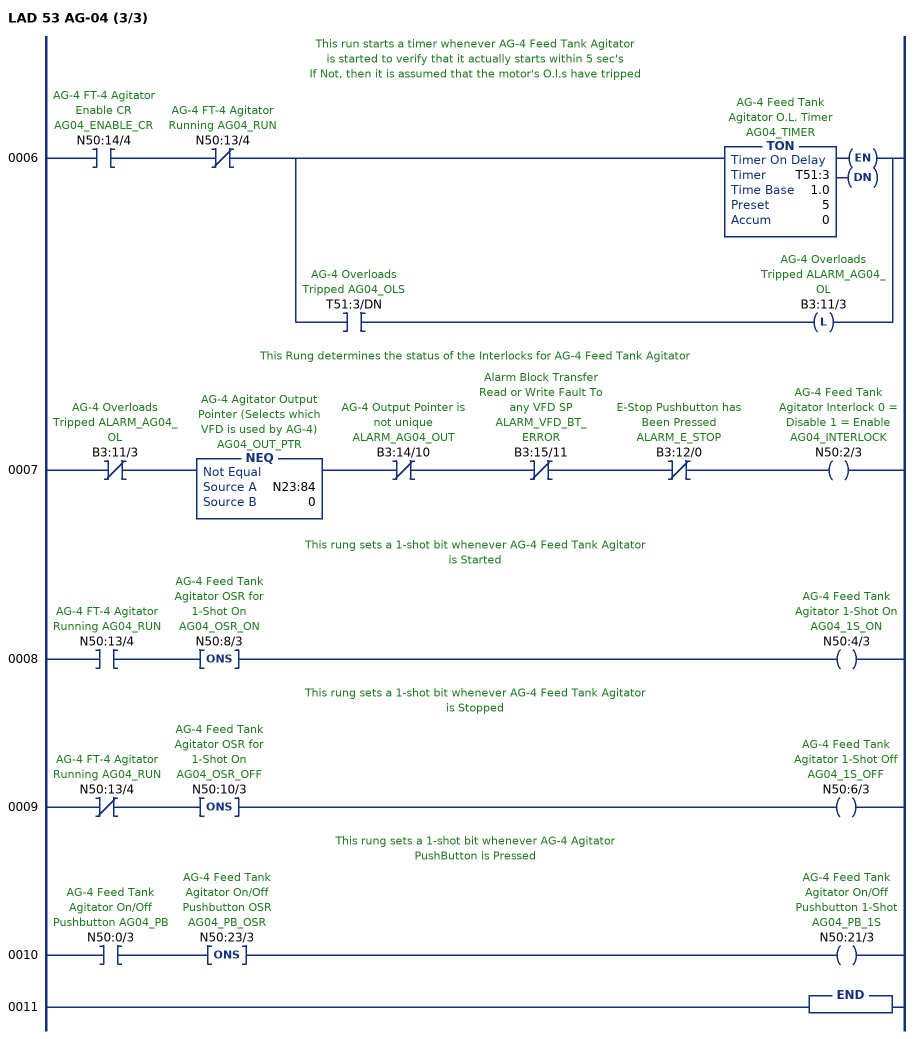
% Rung: 6 %
% This run starts a timer whenever AG-4 Feed Tank Agitator
% is started to verify that it actually starts within 5 sec's
% If Not, then it is assumed that the motor's O.l.s have tripped %
SOR XIC N50:14/4 XIO N50:13/4 BST TON T51:3 1.0 5 0 NXB XIC T51:3/DN OTL B3:11/3 BND EOR
%   N50:14/4  AG04_ENABLE_CR  "AG-4 FT-4 Agitator Enable CR" %
%   N50:13/4  AG04_RUN  "AG-4 FT-4 Agitator Running" %
%   T51:3  AG04_TIMER  "AG-4 Feed Tank Agitator O.L. Timer" %
%   T51:3/DN  AG04_OLS  "AG-4 Overloads Tripped" %
%   B3:11/3  ALARM_AG04_OL  "AG-4 Overloads Tripped" %
% Rung: 7 %
% This Rung determines the status of the Interlocks for AG-4 Feed Tank Agitator %
SOR XIO B3:11/3 NEQ N23:84 0 XIO B3:14/10 XIO B3:15/11 XIO B3:12/0 OTE N50:2/3 EOR
%   B3:11/3  ALARM_AG04_OL  "AG-4 Overloads Tripped" %
%   N23:84  AG04_OUT_PTR  "AG-4 Agitator Output Pointer (Selects which VFD is used by AG-4)" %
%   B3:14/10  ALARM_AG04_OUT  "AG-4 Output Pointer is not unique" %
%   B3:15/11  ALARM_VFD_BT_ERROR  "Alarm Block Transfer Read or Write Fault To any VFD SP" %
%   B3:12/0  ALARM_E_STOP  "E-Stop Pushbutton has Been Pressed" %
%   N50:2/3  AG04_INTERLOCK  "AG-4 Feed Tank Agitator Interlock 0 = Disable 1 = Enable" %
% Rung: 8 %
% This rung sets a 1-shot bit whenever AG-4 Feed Tank Agitator
% is Started %
SOR XIC N50:13/4 OSR N50:8/3 OTE N50:4/3 EOR
%   N50:13/4  AG04_RUN  "AG-4 FT-4 Agitator Running" %
%   N50:8/3  AG04_OSR_ON  "AG-4 Feed Tank Agitator OSR for 1-Shot On" %
%   N50:4/3  AG04_1S_ON  "AG-4 Feed Tank Agitator 1-Shot On" %
% Rung: 9 %
% This rung sets a 1-shot bit whenever AG-4 Feed Tank Agitator
% is Stopped %
SOR XIO N50:13/4 OSR N50:10/3 OTE N50:6/3 EOR
%   N50:13/4  AG04_RUN  "AG-4 FT-4 Agitator Running" %
%   N50:10/3  AG04_OSR_OFF  "AG-4 Feed Tank Agitator OSR for 1-Shot On" %
%   N50:6/3  AG04_1S_OFF  "AG-4 Feed Tank Agitator 1-Shot Off" %
% Rung: 10 %
% This rung sets a 1-shot bit whenever AG-4 Agitator
% PushButton is Pressed %
SOR XIC N50:0/3 OSR N50:23/3 OTE N50:21/3 EOR
%   N50:0/3  AG04_PB  "AG-4 Feed Tank Agitator On/Off Pushbutton" %
%   N50:23/3  AG04_PB_OSR  "AG-4 Feed Tank Agitator On/Off Pushbutton OSR" %
%   N50:21/3  AG04_PB_1S  "AG-4 Feed Tank Agitator On/Off Pushbutton 1-Shot" %
% Rung: 11 %
SOR END EOR

LADDER 56 "VP-09"    % VP-9 Beach-Ross Vacuum Pump Controls %
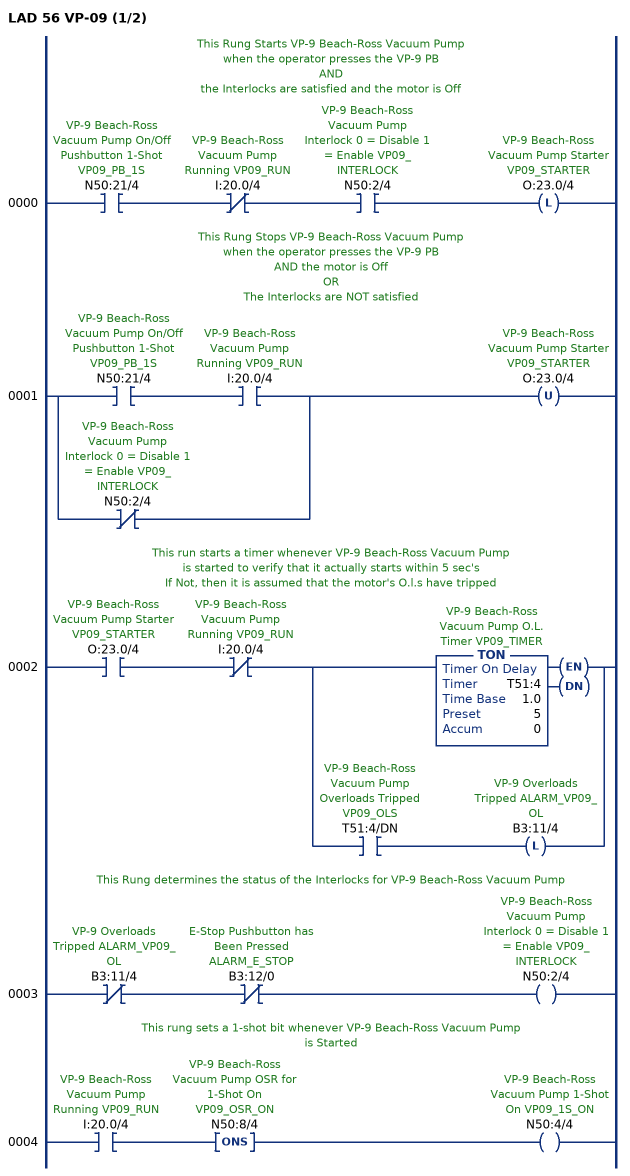
% Rung: 0 %
% This Rung Starts VP-9 Beach-Ross Vacuum Pump
% when the operator presses the VP-9 PB
% AND
% the Interlocks are satisfied and the motor is Off %
SOR XIC N50:21/4 XIO I:20.0/4 XIC N50:2/4 OTL O:23.0/4 EOR
%   N50:21/4  VP09_PB_1S  "VP-9 Beach-Ross Vacuum Pump On/Off Pushbutton 1-Shot" %
%   I:20.0/4  VP09_RUN  "VP-9 Beach-Ross Vacuum Pump Running" %
%   N50:2/4  VP09_INTERLOCK  "VP-9 Beach-Ross Vacuum Pump Interlock 0 = Disable 1 = Enable" %
%   O:23.0/4  VP09_STARTER  "VP-9 Beach-Ross Vacuum Pump Starter" %
% Rung: 1 %
% This Rung Stops VP-9 Beach-Ross Vacuum Pump
% when the operator presses the VP-9 PB
% AND the motor is Off
% OR
% The Interlocks are NOT satisfied %
SOR BST XIC N50:21/4 XIC I:20.0/4 NXB XIO N50:2/4 BND OTU O:23.0/4 EOR
%   N50:21/4  VP09_PB_1S  "VP-9 Beach-Ross Vacuum Pump On/Off Pushbutton 1-Shot" %
%   I:20.0/4  VP09_RUN  "VP-9 Beach-Ross Vacuum Pump Running" %
%   N50:2/4  VP09_INTERLOCK  "VP-9 Beach-Ross Vacuum Pump Interlock 0 = Disable 1 = Enable" %
%   O:23.0/4  VP09_STARTER  "VP-9 Beach-Ross Vacuum Pump Starter" %
% Rung: 2 %
% This run starts a timer whenever VP-9 Beach-Ross Vacuum Pump
% is started to verify that it actually starts within 5 sec's
% If Not, then it is assumed that the motor's O.l.s have tripped %
SOR XIC O:23.0/4 XIO I:20.0/4 BST TON T51:4 1.0 5 0 NXB XIC T51:4/DN OTL B3:11/4 BND EOR
%   O:23.0/4  VP09_STARTER  "VP-9 Beach-Ross Vacuum Pump Starter" %
%   I:20.0/4  VP09_RUN  "VP-9 Beach-Ross Vacuum Pump Running" %
%   T51:4  VP09_TIMER  "VP-9 Beach-Ross Vacuum Pump O.L. Timer" %
%   T51:4/DN  VP09_OLS  "VP-9 Beach-Ross Vacuum Pump Overloads Tripped" %
%   B3:11/4  ALARM_VP09_OL  "VP-9 Overloads Tripped" %
% Rung: 3 %
% This Rung determines the status of the Interlocks for VP-9 Beach-Ross Vacuum Pump %
SOR XIO B3:11/4 XIO B3:12/0 OTE N50:2/4 EOR
%   B3:11/4  ALARM_VP09_OL  "VP-9 Overloads Tripped" %
%   B3:12/0  ALARM_E_STOP  "E-Stop Pushbutton has Been Pressed" %
%   N50:2/4  VP09_INTERLOCK  "VP-9 Beach-Ross Vacuum Pump Interlock 0 = Disable 1 = Enable" %
% Rung: 4 %
% This rung sets a 1-shot bit whenever VP-9 Beach-Ross Vacuum Pump
% is Started %
SOR XIC I:20.0/4 OSR N50:8/4 OTE N50:4/4 EOR
%   I:20.0/4  VP09_RUN  "VP-9 Beach-Ross Vacuum Pump Running" %
%   N50:8/4  VP09_OSR_ON  "VP-9 Beach-Ross Vacuum Pump OSR for 1-Shot On" %
%   N50:4/4  VP09_1S_ON  "VP-9 Beach-Ross Vacuum Pump 1-Shot On" %

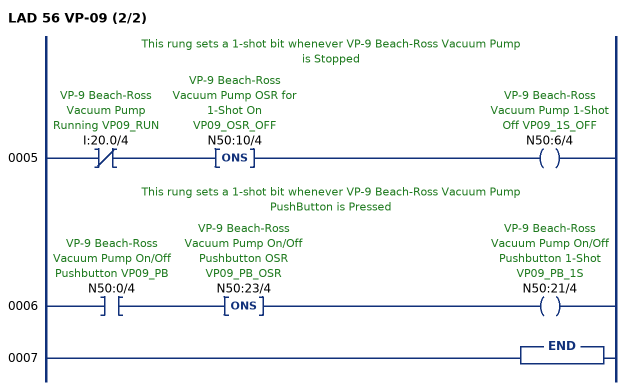
% Rung: 5 %
% This rung sets a 1-shot bit whenever VP-9 Beach-Ross Vacuum Pump
% is Stopped %
SOR XIO I:20.0/4 OSR N50:10/4 OTE N50:6/4 EOR
%   I:20.0/4  VP09_RUN  "VP-9 Beach-Ross Vacuum Pump Running" %
%   N50:10/4  VP09_OSR_OFF  "VP-9 Beach-Ross Vacuum Pump OSR for 1-Shot On" %
%   N50:6/4  VP09_1S_OFF  "VP-9 Beach-Ross Vacuum Pump 1-Shot Off" %
% Rung: 6 %
% This rung sets a 1-shot bit whenever VP-9 Beach-Ross Vacuum Pump
% PushButton is Pressed %
SOR XIC N50:0/4 OSR N50:23/4 OTE N50:21/4 EOR
%   N50:0/4  VP09_PB  "VP-9 Beach-Ross Vacuum Pump On/Off Pushbutton" %
%   N50:23/4  VP09_PB_OSR  "VP-9 Beach-Ross Vacuum Pump On/Off Pushbutton OSR" %
%   N50:21/4  VP09_PB_1S  "VP-9 Beach-Ross Vacuum Pump On/Off Pushbutton 1-Shot" %
% Rung: 7 %
SOR END EOR

LADDER 57 "VP-10"    % VP-10 Kinney Vacuum Pump Controls %
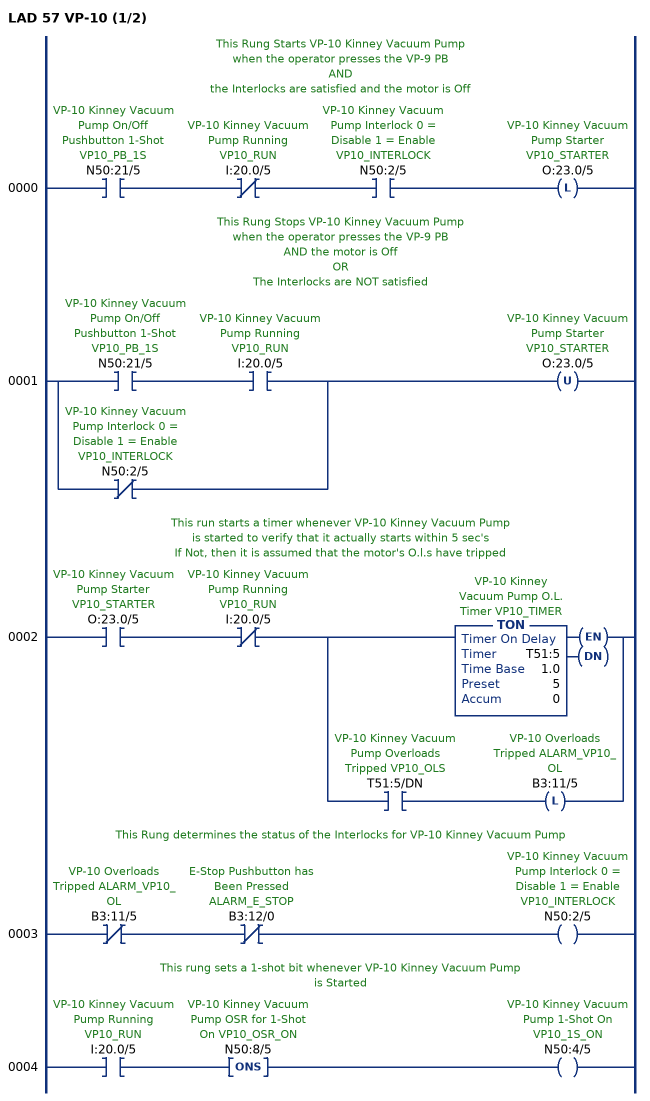
% Rung: 0 %
% This Rung Starts VP-10 Kinney Vacuum Pump
% when the operator presses the VP-9 PB
% AND
% the Interlocks are satisfied and the motor is Off %
SOR XIC N50:21/5 XIO I:20.0/5 XIC N50:2/5 OTL O:23.0/5 EOR
%   N50:21/5  VP10_PB_1S  "VP-10 Kinney Vacuum Pump On/Off Pushbutton 1-Shot" %
%   I:20.0/5  VP10_RUN  "VP-10 Kinney Vacuum Pump Running" %
%   N50:2/5  VP10_INTERLOCK  "VP-10 Kinney Vacuum Pump Interlock 0 = Disable 1 = Enable" %
%   O:23.0/5  VP10_STARTER  "VP-10 Kinney Vacuum Pump Starter" %
% Rung: 1 %
% This Rung Stops VP-10 Kinney Vacuum Pump
% when the operator presses the VP-9 PB
% AND the motor is Off
% OR
% The Interlocks are NOT satisfied %
SOR BST XIC N50:21/5 XIC I:20.0/5 NXB XIO N50:2/5 BND OTU O:23.0/5 EOR
%   N50:21/5  VP10_PB_1S  "VP-10 Kinney Vacuum Pump On/Off Pushbutton 1-Shot" %
%   I:20.0/5  VP10_RUN  "VP-10 Kinney Vacuum Pump Running" %
%   N50:2/5  VP10_INTERLOCK  "VP-10 Kinney Vacuum Pump Interlock 0 = Disable 1 = Enable" %
%   O:23.0/5  VP10_STARTER  "VP-10 Kinney Vacuum Pump Starter" %
% Rung: 2 %
% This run starts a timer whenever VP-10 Kinney Vacuum Pump
% is started to verify that it actually starts within 5 sec's
% If Not, then it is assumed that the motor's O.l.s have tripped %
SOR XIC O:23.0/5 XIO I:20.0/5 BST TON T51:5 1.0 5 0 NXB XIC T51:5/DN OTL B3:11/5 BND EOR
%   O:23.0/5  VP10_STARTER  "VP-10 Kinney Vacuum Pump Starter" %
%   I:20.0/5  VP10_RUN  "VP-10 Kinney Vacuum Pump Running" %
%   T51:5  VP10_TIMER  "VP-10 Kinney Vacuum Pump O.L. Timer" %
%   T51:5/DN  VP10_OLS  "VP-10 Kinney Vacuum Pump Overloads Tripped" %
%   B3:11/5  ALARM_VP10_OL  "VP-10 Overloads Tripped" %
% Rung: 3 %
% This Rung determines the status of the Interlocks for VP-10 Kinney Vacuum Pump %
SOR XIO B3:11/5 XIO B3:12/0 OTE N50:2/5 EOR
%   B3:11/5  ALARM_VP10_OL  "VP-10 Overloads Tripped" %
%   B3:12/0  ALARM_E_STOP  "E-Stop Pushbutton has Been Pressed" %
%   N50:2/5  VP10_INTERLOCK  "VP-10 Kinney Vacuum Pump Interlock 0 = Disable 1 = Enable" %
% Rung: 4 %
% This rung sets a 1-shot bit whenever VP-10 Kinney Vacuum Pump
% is Started %
SOR XIC I:20.0/5 OSR N50:8/5 OTE N50:4/5 EOR
%   I:20.0/5  VP10_RUN  "VP-10 Kinney Vacuum Pump Running" %
%   N50:8/5  VP10_OSR_ON  "VP-10 Kinney Vacuum Pump OSR for 1-Shot On" %
%   N50:4/5  VP10_1S_ON  "VP-10 Kinney Vacuum Pump 1-Shot On" %

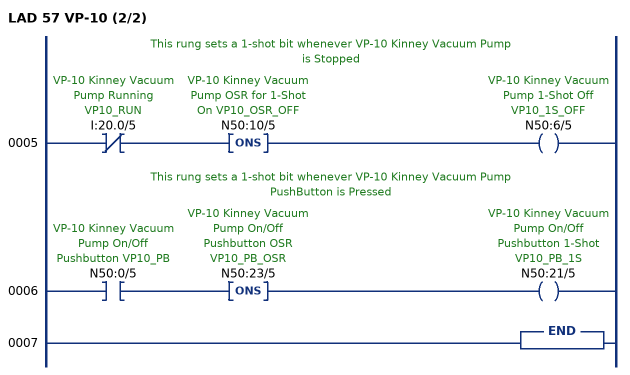
% Rung: 5 %
% This rung sets a 1-shot bit whenever VP-10 Kinney Vacuum Pump
% is Stopped %
SOR XIO I:20.0/5 OSR N50:10/5 OTE N50:6/5 EOR
%   I:20.0/5  VP10_RUN  "VP-10 Kinney Vacuum Pump Running" %
%   N50:10/5  VP10_OSR_OFF  "VP-10 Kinney Vacuum Pump OSR for 1-Shot On" %
%   N50:6/5  VP10_1S_OFF  "VP-10 Kinney Vacuum Pump 1-Shot Off" %
% Rung: 6 %
% This rung sets a 1-shot bit whenever VP-10 Kinney Vacuum Pump
% PushButton is Pressed %
SOR XIC N50:0/5 OSR N50:23/5 OTE N50:21/5 EOR
%   N50:0/5  VP10_PB  "VP-10 Kinney Vacuum Pump On/Off Pushbutton" %
%   N50:23/5  VP10_PB_OSR  "VP-10 Kinney Vacuum Pump On/Off Pushbutton OSR" %
%   N50:21/5  VP10_PB_1S  "VP-10 Kinney Vacuum Pump On/Off Pushbutton 1-Shot" %
% Rung: 7 %
SOR END EOR

LADDER 60 "PU-11"    % PU-11 Tempered Water Loop No-1 Circ Pump Controls %
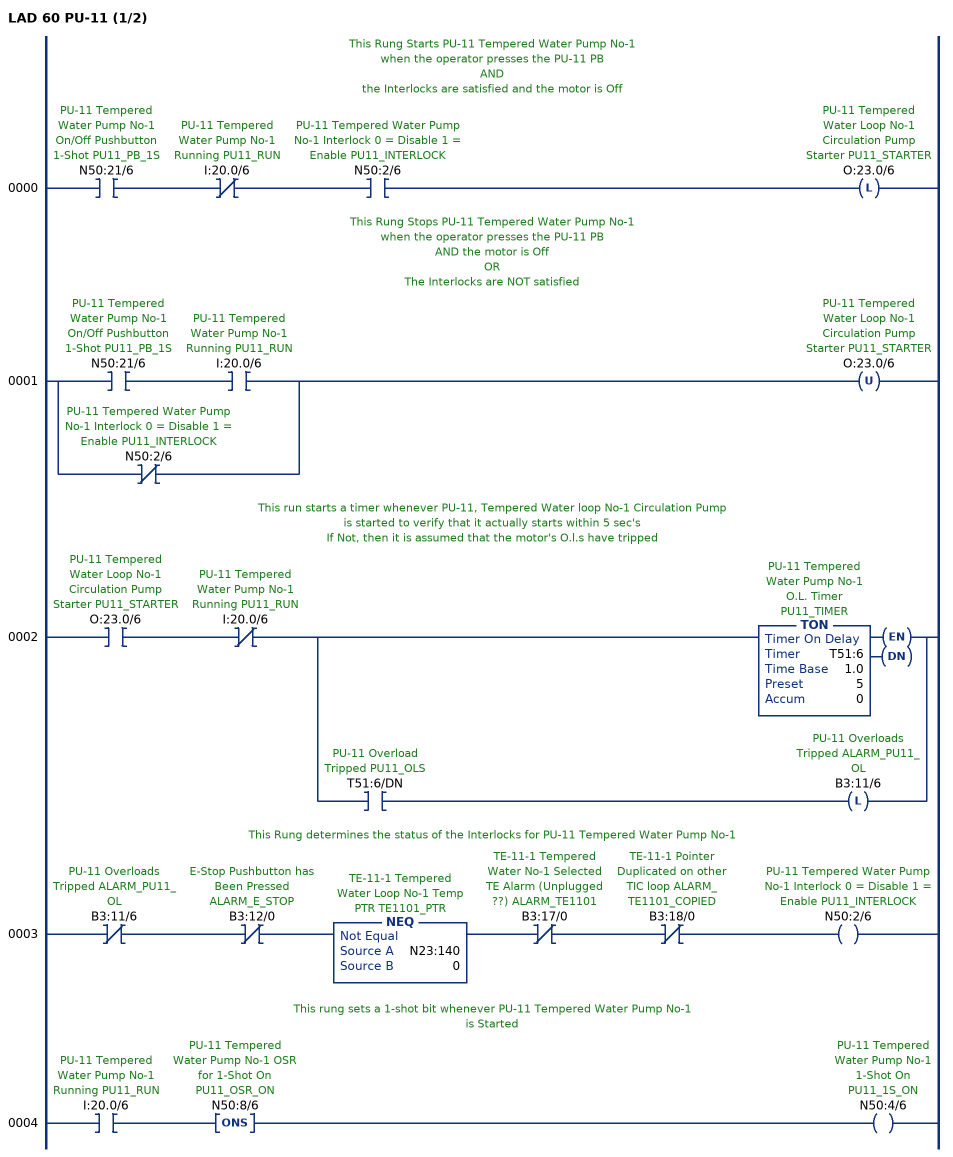
% Rung: 0 %
% This Rung Starts PU-11 Tempered Water Pump No-1
% when the operator presses the PU-11 PB
% AND
% the Interlocks are satisfied and the motor is Off %
SOR XIC N50:21/6 XIO I:20.0/6 XIC N50:2/6 OTL O:23.0/6 EOR
%   N50:21/6  PU11_PB_1S  "PU-11 Tempered Water Pump No-1 On/Off Pushbutton 1-Shot" %
%   I:20.0/6  PU11_RUN  "PU-11 Tempered Water Pump No-1 Running" %
%   N50:2/6  PU11_INTERLOCK  "PU-11 Tempered Water Pump No-1 Interlock 0 = Disable 1 = Enable" %
%   O:23.0/6  PU11_STARTER  "PU-11 Tempered Water Loop No-1 Circulation Pump Starter" %
% Rung: 1 %
% This Rung Stops PU-11 Tempered Water Pump No-1
% when the operator presses the PU-11 PB
% AND the motor is Off
% OR
% The Interlocks are NOT satisfied %
SOR BST XIC N50:21/6 XIC I:20.0/6 NXB XIO N50:2/6 BND OTU O:23.0/6 EOR
%   N50:21/6  PU11_PB_1S  "PU-11 Tempered Water Pump No-1 On/Off Pushbutton 1-Shot" %
%   I:20.0/6  PU11_RUN  "PU-11 Tempered Water Pump No-1 Running" %
%   N50:2/6  PU11_INTERLOCK  "PU-11 Tempered Water Pump No-1 Interlock 0 = Disable 1 = Enable" %
%   O:23.0/6  PU11_STARTER  "PU-11 Tempered Water Loop No-1 Circulation Pump Starter" %
% Rung: 2 %
% This run starts a timer whenever PU-11, Tempered Water loop No-1 Circulation Pump
% is started to verify that it actually starts within 5 sec's
% If Not, then it is assumed that the motor's O.l.s have tripped %
SOR XIC O:23.0/6 XIO I:20.0/6 BST TON T51:6 1.0 5 0 NXB XIC T51:6/DN OTL B3:11/6 BND EOR
%   O:23.0/6  PU11_STARTER  "PU-11 Tempered Water Loop No-1 Circulation Pump Starter" %
%   I:20.0/6  PU11_RUN  "PU-11 Tempered Water Pump No-1 Running" %
%   T51:6  PU11_TIMER  "PU-11 Tempered Water Pump No-1 O.L. Timer" %
%   T51:6/DN  PU11_OLS  "PU-11 Overload Tripped" %
%   B3:11/6  ALARM_PU11_OL  "PU-11 Overloads Tripped" %
% Rung: 3 %
% This Rung determines the status of the Interlocks for PU-11 Tempered Water Pump No-1 %
SOR XIO B3:11/6 XIO B3:12/0 NEQ N23:140 0 XIO B3:17/0 XIO B3:18/0 OTE N50:2/6 EOR
%   B3:11/6  ALARM_PU11_OL  "PU-11 Overloads Tripped" %
%   B3:12/0  ALARM_E_STOP  "E-Stop Pushbutton has Been Pressed" %
%   N23:140  TE1101_PTR  "TE-11-1 Tempered Water Loop No-1 Temp PTR" %
%   B3:17/0  ALARM_TE1101  "TE-11-1 Tempered Water No-1 Selected TE Alarm (Unplugged ??)" %
%   B3:18/0  ALARM_TE1101_COPIED  "TE-11-1 Pointer Duplicated on other TIC loop" %
%   N50:2/6  PU11_INTERLOCK  "PU-11 Tempered Water Pump No-1 Interlock 0 = Disable 1 = Enable" %
% Rung: 4 %
% This rung sets a 1-shot bit whenever PU-11 Tempered Water Pump No-1
% is Started %
SOR XIC I:20.0/6 OSR N50:8/6 OTE N50:4/6 EOR
%   I:20.0/6  PU11_RUN  "PU-11 Tempered Water Pump No-1 Running" %
%   N50:8/6  PU11_OSR_ON  "PU-11 Tempered Water Pump No-1 OSR for 1-Shot On" %
%   N50:4/6  PU11_1S_ON  "PU-11 Tempered Water Pump No-1 1-Shot On" %

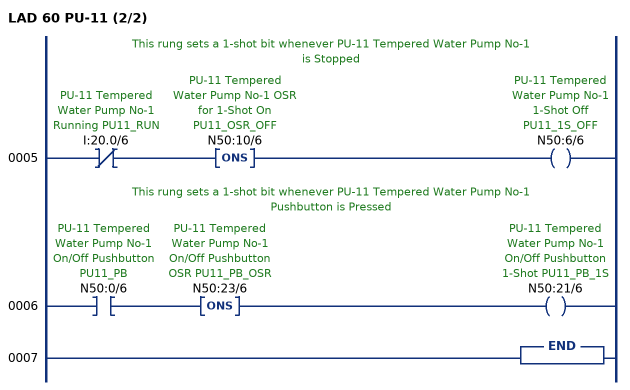
% Rung: 5 %
% This rung sets a 1-shot bit whenever PU-11 Tempered Water Pump No-1
% is Stopped %
SOR XIO I:20.0/6 OSR N50:10/6 OTE N50:6/6 EOR
%   I:20.0/6  PU11_RUN  "PU-11 Tempered Water Pump No-1 Running" %
%   N50:10/6  PU11_OSR_OFF  "PU-11 Tempered Water Pump No-1 OSR for 1-Shot On" %
%   N50:6/6  PU11_1S_OFF  "PU-11 Tempered Water Pump No-1 1-Shot Off" %
% Rung: 6 %
% This rung sets a 1-shot bit whenever PU-11 Tempered Water Pump No-1
% Pushbutton is Pressed %
SOR XIC N50:0/6 OSR N50:23/6 OTE N50:21/6 EOR
%   N50:0/6  PU11_PB  "PU-11 Tempered Water Pump No-1 On/Off Pushbutton" %
%   N50:23/6  PU11_PB_OSR  "PU-11 Tempered Water Pump No-1 On/Off Pushbutton OSR" %
%   N50:21/6  PU11_PB_1S  "PU-11 Tempered Water Pump No-1 On/Off Pushbutton 1-Shot" %
% Rung: 7 %
SOR END EOR

LADDER 61 "PU-12"    % PU-12 Tempered Water Loop No-2 Circ Pump Controls %
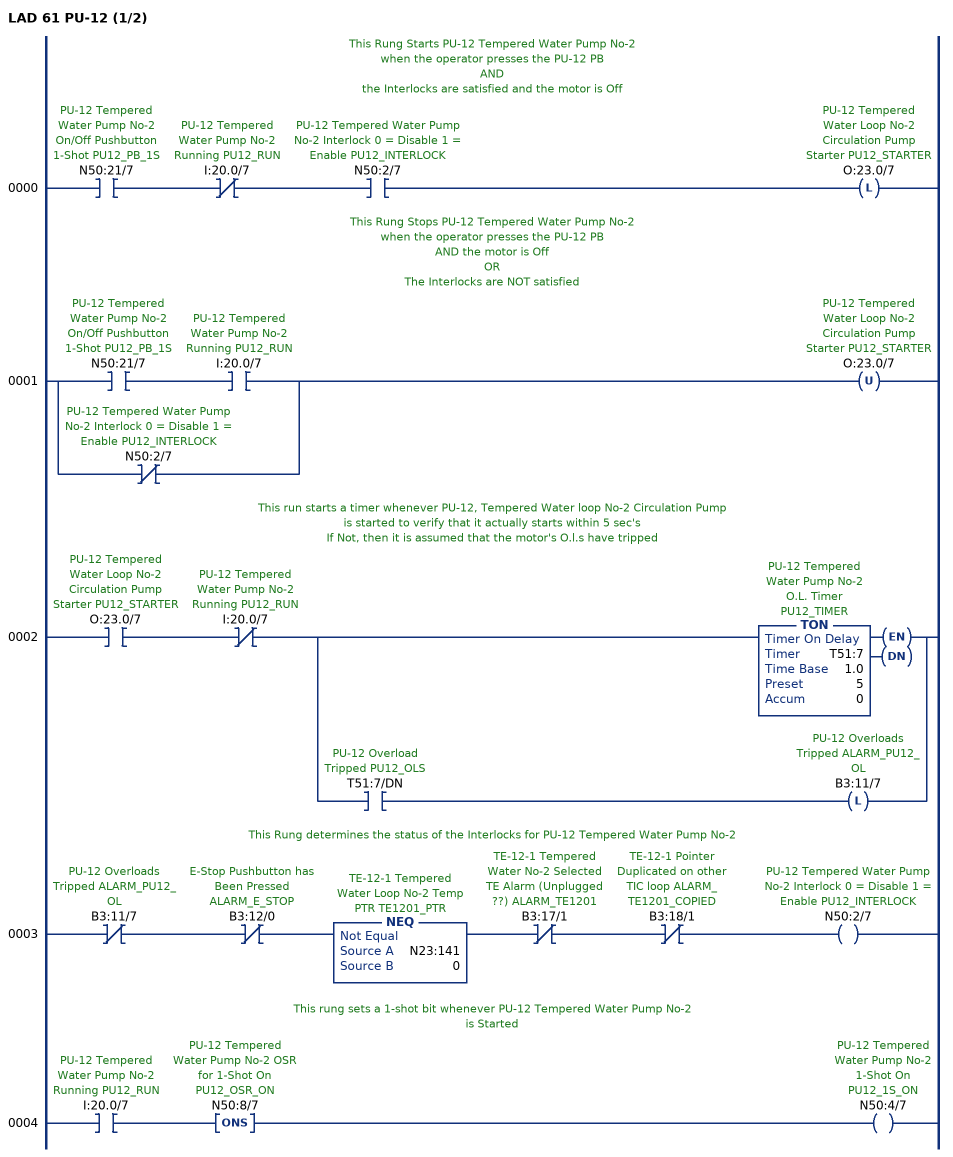
% Rung: 0 %
% This Rung Starts PU-12 Tempered Water Pump No-2
% when the operator presses the PU-12 PB
% AND
% the Interlocks are satisfied and the motor is Off %
SOR XIC N50:21/7 XIO I:20.0/7 XIC N50:2/7 OTL O:23.0/7 EOR
%   N50:21/7  PU12_PB_1S  "PU-12 Tempered Water Pump No-2 On/Off Pushbutton 1-Shot" %
%   I:20.0/7  PU12_RUN  "PU-12 Tempered Water Pump No-2 Running" %
%   N50:2/7  PU12_INTERLOCK  "PU-12 Tempered Water Pump No-2 Interlock 0 = Disable 1 = Enable" %
%   O:23.0/7  PU12_STARTER  "PU-12 Tempered Water Loop No-2 Circulation Pump Starter" %
% Rung: 1 %
% This Rung Stops PU-12 Tempered Water Pump No-2
% when the operator presses the PU-12 PB
% AND the motor is Off
% OR
% The Interlocks are NOT satisfied %
SOR BST XIC N50:21/7 XIC I:20.0/7 NXB XIO N50:2/7 BND OTU O:23.0/7 EOR
%   N50:21/7  PU12_PB_1S  "PU-12 Tempered Water Pump No-2 On/Off Pushbutton 1-Shot" %
%   I:20.0/7  PU12_RUN  "PU-12 Tempered Water Pump No-2 Running" %
%   N50:2/7  PU12_INTERLOCK  "PU-12 Tempered Water Pump No-2 Interlock 0 = Disable 1 = Enable" %
%   O:23.0/7  PU12_STARTER  "PU-12 Tempered Water Loop No-2 Circulation Pump Starter" %
% Rung: 2 %
% This run starts a timer whenever PU-12, Tempered Water loop No-2 Circulation Pump
% is started to verify that it actually starts within 5 sec's
% If Not, then it is assumed that the motor's O.l.s have tripped %
SOR XIC O:23.0/7 XIO I:20.0/7 BST TON T51:7 1.0 5 0 NXB XIC T51:7/DN OTL B3:11/7 BND EOR
%   O:23.0/7  PU12_STARTER  "PU-12 Tempered Water Loop No-2 Circulation Pump Starter" %
%   I:20.0/7  PU12_RUN  "PU-12 Tempered Water Pump No-2 Running" %
%   T51:7  PU12_TIMER  "PU-12 Tempered Water Pump No-2 O.L. Timer" %
%   T51:7/DN  PU12_OLS  "PU-12 Overload Tripped" %
%   B3:11/7  ALARM_PU12_OL  "PU-12 Overloads Tripped" %
% Rung: 3 %
% This Rung determines the status of the Interlocks for PU-12 Tempered Water Pump No-2 %
SOR XIO B3:11/7 XIO B3:12/0 NEQ N23:141 0 XIO B3:17/1 XIO B3:18/1 OTE N50:2/7 EOR
%   B3:11/7  ALARM_PU12_OL  "PU-12 Overloads Tripped" %
%   B3:12/0  ALARM_E_STOP  "E-Stop Pushbutton has Been Pressed" %
%   N23:141  TE1201_PTR  "TE-12-1 Tempered Water Loop No-2 Temp PTR" %
%   B3:17/1  ALARM_TE1201  "TE-12-1 Tempered Water No-2 Selected TE Alarm (Unplugged ??)" %
%   B3:18/1  ALARM_TE1201_COPIED  "TE-12-1 Pointer Duplicated on other TIC loop" %
%   N50:2/7  PU12_INTERLOCK  "PU-12 Tempered Water Pump No-2 Interlock 0 = Disable 1 = Enable" %
% Rung: 4 %
% This rung sets a 1-shot bit whenever PU-12 Tempered Water Pump No-2
% is Started %
SOR XIC I:20.0/7 OSR N50:8/7 OTE N50:4/7 EOR
%   I:20.0/7  PU12_RUN  "PU-12 Tempered Water Pump No-2 Running" %
%   N50:8/7  PU12_OSR_ON  "PU-12 Tempered Water Pump No-2 OSR for 1-Shot On" %
%   N50:4/7  PU12_1S_ON  "PU-12 Tempered Water Pump No-2 1-Shot On" %

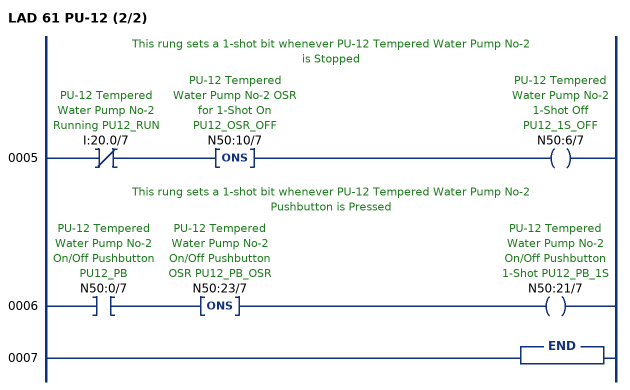
% Rung: 5 %
% This rung sets a 1-shot bit whenever PU-12 Tempered Water Pump No-2
% is Stopped %
SOR XIO I:20.0/7 OSR N50:10/7 OTE N50:6/7 EOR
%   I:20.0/7  PU12_RUN  "PU-12 Tempered Water Pump No-2 Running" %
%   N50:10/7  PU12_OSR_OFF  "PU-12 Tempered Water Pump No-2 OSR for 1-Shot On" %
%   N50:6/7  PU12_1S_OFF  "PU-12 Tempered Water Pump No-2 1-Shot Off" %
% Rung: 6 %
% This rung sets a 1-shot bit whenever PU-12 Tempered Water Pump No-2
% Pushbutton is Pressed %
SOR XIC N50:0/7 OSR N50:23/7 OTE N50:21/7 EOR
%   N50:0/7  PU12_PB  "PU-12 Tempered Water Pump No-2 On/Off Pushbutton" %
%   N50:23/7  PU12_PB_OSR  "PU-12 Tempered Water Pump No-2 On/Off Pushbutton OSR" %
%   N50:21/7  PU12_PB_1S  "PU-12 Tempered Water Pump No-2 On/Off Pushbutton 1-Shot" %
% Rung: 7 %
SOR END EOR

LADDER 62 "PU-15"    % PU-15 Tempered Oil Loop No-1 Circ Pump Controls %
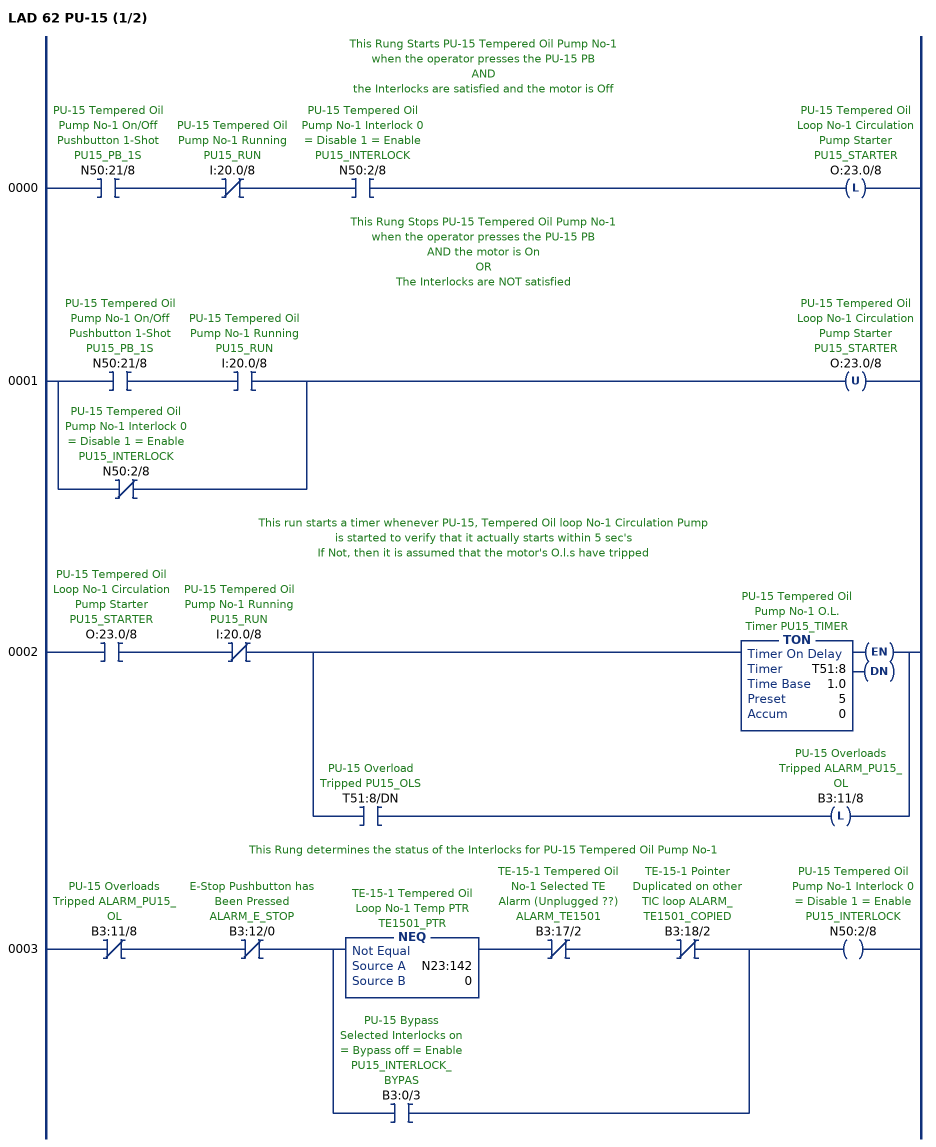
% Rung: 0 %
% This Rung Starts PU-15 Tempered Oil Pump No-1
% when the operator presses the PU-15 PB
% AND
% the Interlocks are satisfied and the motor is Off %
SOR XIC N50:21/8 XIO I:20.0/8 XIC N50:2/8 OTL O:23.0/8 EOR
%   N50:21/8  PU15_PB_1S  "PU-15 Tempered Oil Pump No-1 On/Off Pushbutton 1-Shot" %
%   I:20.0/8  PU15_RUN  "PU-15 Tempered Oil Pump No-1 Running" %
%   N50:2/8  PU15_INTERLOCK  "PU-15 Tempered Oil Pump No-1 Interlock 0 = Disable 1 = Enable" %
%   O:23.0/8  PU15_STARTER  "PU-15 Tempered Oil Loop No-1 Circulation Pump Starter" %
% Rung: 1 %
% This Rung Stops PU-15 Tempered Oil Pump No-1
% when the operator presses the PU-15 PB
% AND the motor is On
% OR
% The Interlocks are NOT satisfied %
SOR BST XIC N50:21/8 XIC I:20.0/8 NXB XIO N50:2/8 BND OTU O:23.0/8 EOR
%   N50:21/8  PU15_PB_1S  "PU-15 Tempered Oil Pump No-1 On/Off Pushbutton 1-Shot" %
%   I:20.0/8  PU15_RUN  "PU-15 Tempered Oil Pump No-1 Running" %
%   N50:2/8  PU15_INTERLOCK  "PU-15 Tempered Oil Pump No-1 Interlock 0 = Disable 1 = Enable" %
%   O:23.0/8  PU15_STARTER  "PU-15 Tempered Oil Loop No-1 Circulation Pump Starter" %
% Rung: 2 %
% This run starts a timer whenever PU-15, Tempered Oil loop No-1 Circulation Pump
% is started to verify that it actually starts within 5 sec's
% If Not, then it is assumed that the motor's O.l.s have tripped %
SOR XIC O:23.0/8 XIO I:20.0/8 BST TON T51:8 1.0 5 0 NXB XIC T51:8/DN OTL B3:11/8 BND EOR
%   O:23.0/8  PU15_STARTER  "PU-15 Tempered Oil Loop No-1 Circulation Pump Starter" %
%   I:20.0/8  PU15_RUN  "PU-15 Tempered Oil Pump No-1 Running" %
%   T51:8  PU15_TIMER  "PU-15 Tempered Oil Pump No-1 O.L. Timer" %
%   T51:8/DN  PU15_OLS  "PU-15 Overload Tripped" %
%   B3:11/8  ALARM_PU15_OL  "PU-15 Overloads Tripped" %
% Rung: 3 %
% This Rung determines the status of the Interlocks for PU-15 Tempered Oil Pump No-1 %
SOR XIO B3:11/8 XIO B3:12/0 BST NEQ N23:142 0 XIO B3:17/2 XIO B3:18/2 NXB XIC B3:0/3 BND OTE N50:2/8 EOR
%   B3:11/8  ALARM_PU15_OL  "PU-15 Overloads Tripped" %
%   B3:12/0  ALARM_E_STOP  "E-Stop Pushbutton has Been Pressed" %
%   N23:142  TE1501_PTR  "TE-15-1 Tempered Oil Loop No-1 Temp PTR" %
%   B3:17/2  ALARM_TE1501  "TE-15-1 Tempered Oil No-1 Selected TE Alarm (Unplugged ??)" %
%   B3:18/2  ALARM_TE1501_COPIED  "TE-15-1 Pointer Duplicated on other TIC loop" %
%   B3:0/3  PU15_INTERLOCK_BYPAS  "PU-15 Bypass Selected Interlocks on = Bypass off = Enable" %
%   N50:2/8  PU15_INTERLOCK  "PU-15 Tempered Oil Pump No-1 Interlock 0 = Disable 1 = Enable" %

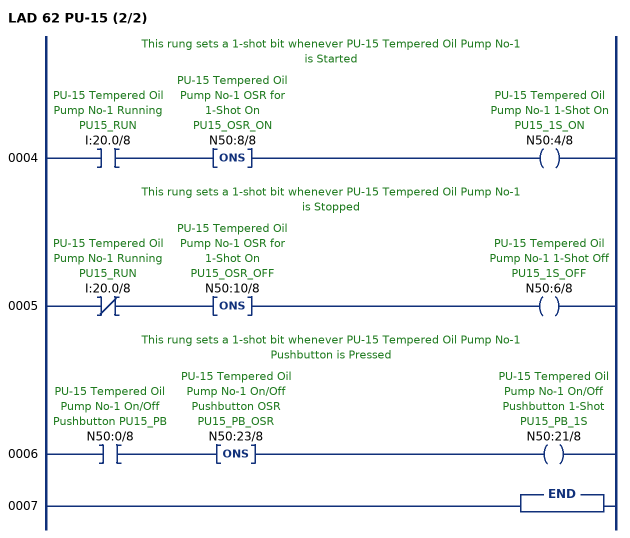
% Rung: 4 %
% This rung sets a 1-shot bit whenever PU-15 Tempered Oil Pump No-1
% is Started %
SOR XIC I:20.0/8 OSR N50:8/8 OTE N50:4/8 EOR
%   I:20.0/8  PU15_RUN  "PU-15 Tempered Oil Pump No-1 Running" %
%   N50:8/8  PU15_OSR_ON  "PU-15 Tempered Oil Pump No-1 OSR for 1-Shot On" %
%   N50:4/8  PU15_1S_ON  "PU-15 Tempered Oil Pump No-1 1-Shot On" %
% Rung: 5 %
% This rung sets a 1-shot bit whenever PU-15 Tempered Oil Pump No-1
% is Stopped %
SOR XIO I:20.0/8 OSR N50:10/8 OTE N50:6/8 EOR
%   I:20.0/8  PU15_RUN  "PU-15 Tempered Oil Pump No-1 Running" %
%   N50:10/8  PU15_OSR_OFF  "PU-15 Tempered Oil Pump No-1 OSR for 1-Shot On" %
%   N50:6/8  PU15_1S_OFF  "PU-15 Tempered Oil Pump No-1 1-Shot Off" %
% Rung: 6 %
% This rung sets a 1-shot bit whenever PU-15 Tempered Oil Pump No-1
% Pushbutton is Pressed %
SOR XIC N50:0/8 OSR N50:23/8 OTE N50:21/8 EOR
%   N50:0/8  PU15_PB  "PU-15 Tempered Oil Pump No-1 On/Off Pushbutton" %
%   N50:23/8  PU15_PB_OSR  "PU-15 Tempered Oil Pump No-1 On/Off Pushbutton OSR" %
%   N50:21/8  PU15_PB_1S  "PU-15 Tempered Oil Pump No-1 On/Off Pushbutton 1-Shot" %
% Rung: 7 %
SOR END EOR

LADDER 63 "EV-20"    % EV-20 Rotor Drive VFD Controls %
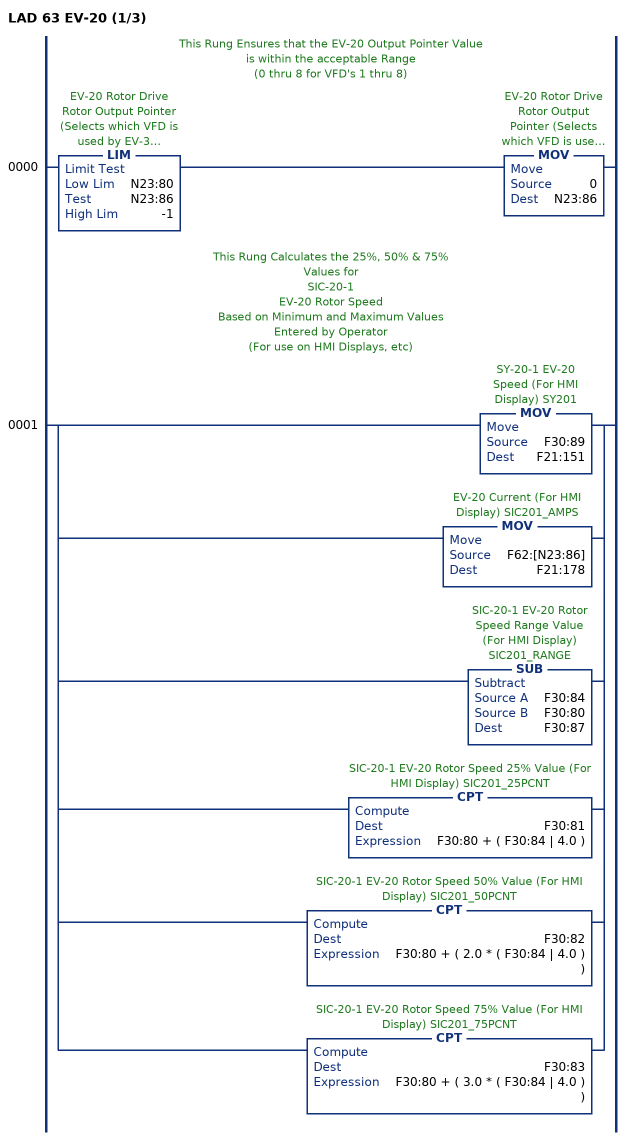
% Rung: 0 %
% This Rung Ensures that the EV-20 Output Pointer Value
% is within the acceptable Range
% (0 thru 8 for VFD's 1 thru 8) %
SOR LIM N23:80 N23:86 -1 MOV 0 N23:86 EOR
%   N23:80  MAX_VFD_ALLOWED_1  "Maximum Number of VFDs Available Plus 1" %
%   N23:86  EV20_OUT_PTR  "EV-20 Rotor Drive Rotor Output Pointer (Selects which VFD is used by EV-3)" %
% Rung: 1 %
% This Rung Calculates the 25%, 50% & 75%
% Values for
% SIC-20-1
% EV-20 Rotor Speed
% Based on Minimum and Maximum Values
% Entered by Operator
% (For use on HMI Displays, etc) %
SOR BST MOV F30:89 F21:151 NXB MOV F62:[N23:86] F21:178 NXB SUB F30:84 F30:80 F30:87 NXB CPT F30:81 " F30:80 + ( F30:84 | 4.0 ) " NXB CPT F30:82 " F30:80 + ( 2.0 * ( F30:84 | 4.0 ) ) " NXB CPT F30:83 " F30:80 + ( 3.0 * ( F30:84 | 4.0 ) ) " BND EOR
%   F30:89  SIC201_SP_FP  "SIC-20-1 EV-20 Rotor Speed Setpoint Value (For HMI Display)" %
%   F21:151  SY201  "SY-20-1 EV-20 Speed (For HMI Display)" %
%   N23:86  EV20_OUT_PTR  "EV-20 Rotor Drive Rotor Output Pointer (Selects which VFD is used by EV-3)" %
%   F21:178  SIC201_AMPS  "EV-20 Current (For HMI Display)" %
%   F30:84  SIC201_MAX  "SIC-20-1 EV-20 Rotor Speed 100% Value (For HMI Display)" %
%   F30:80  SIC201_MIN  "SIC-20-1 EV-20 Rotor Speed 0% Value (For HMI Display)" %
%   F30:87  SIC201_RANGE  "SIC-20-1 EV-20 Rotor Speed Range Value (For HMI Display)" %
%   F30:81  SIC201_25PCNT  "SIC-20-1 EV-20 Rotor Speed 25% Value (For HMI Display)" %
%   F30:82  SIC201_50PCNT  "SIC-20-1 EV-20 Rotor Speed 50% Value (For HMI Display)" %
%   F30:83  SIC201_75PCNT  "SIC-20-1 EV-20 Rotor Speed 75% Value (For HMI Display)" %

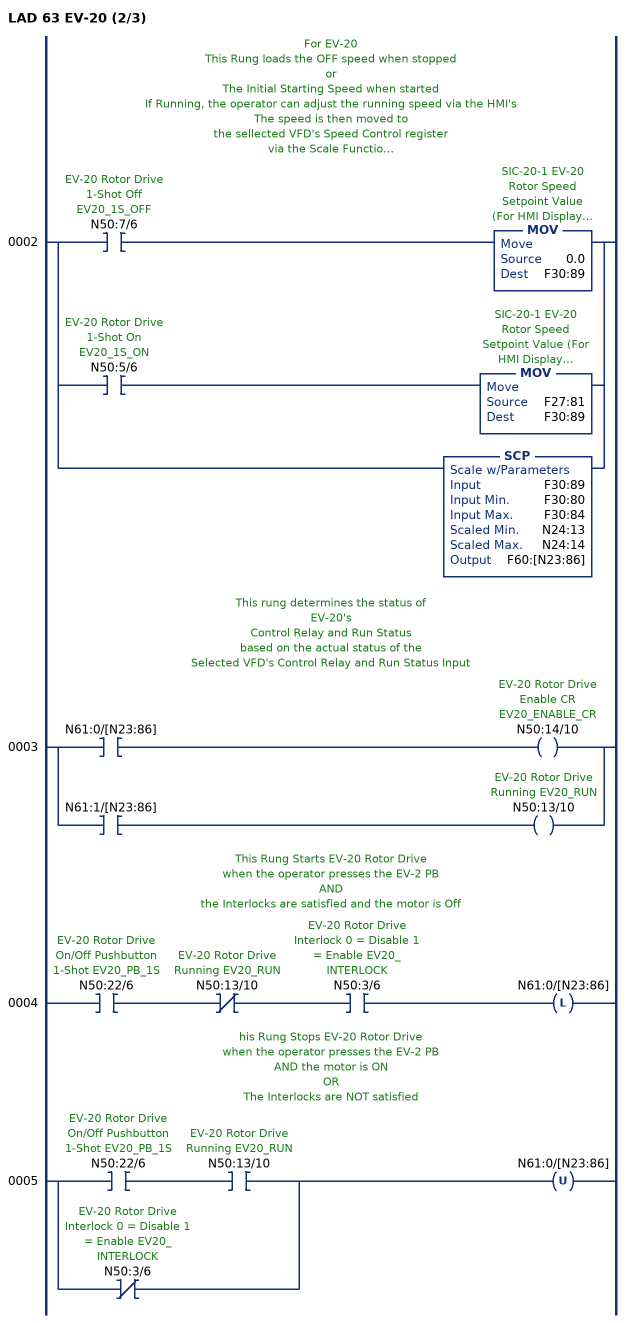
% Rung: 2 %
% For EV-20
% This Rung loads the OFF speed when stopped
% or
% The Initial Starting Speed when started
% If Running, the operator can adjust the running speed via the HMI's
% The speed is then moved to
% the sellected VFD's Speed Control register
% via the Scale Function
% to actually adjust the VFD's Speed %
SOR BST XIC N50:7/6 MOV 0.0 F30:89 NXB XIC N50:5/6 MOV F27:81 F30:89 NXB SCP F30:89 F30:80 F30:84 N24:13 N24:14 F60:[N23:86] BND EOR
%   N50:7/6  EV20_1S_OFF  "EV-20 Rotor Drive 1-Shot Off" %
%   F30:89  SIC201_SP_FP  "SIC-20-1 EV-20 Rotor Speed Setpoint Value (For HMI Display)" %
%   N50:5/6  EV20_1S_ON  "EV-20 Rotor Drive 1-Shot On" %
%   F27:81  SIC201_INIT_SP  "SY-20-1 Initial Speed Setpoint (RPM)" %
%   F30:80  SIC201_MIN  "SIC-20-1 EV-20 Rotor Speed 0% Value (For HMI Display)" %
%   F30:84  SIC201_MAX  "SIC-20-1 EV-20 Rotor Speed 100% Value (For HMI Display)" %
%   N24:13  AO_MIN_OE4  "Analog Output Minimum Value Generates 4 mA DC (To OE4 AO Module)" %
%   N24:14  AO_MAX_OE4  "Analog Output Maximum Value Generates 20 mA DC (To OE4 AO Module)" %
%   N23:86  EV20_OUT_PTR  "EV-20 Rotor Drive Rotor Output Pointer (Selects which VFD is used by EV-3)" %
% Rung: 3 %
% This rung determines the status of
% EV-20's
% Control Relay and Run Status
% based on the actual status of the
% Selected VFD's Control Relay and Run Status Input %
SOR BST XIC N61:0/[N23:86] OTE N50:14/10 NXB XIC N61:1/[N23:86] OTE N50:13/10 BND EOR
%   N61:0  VFD_ENABLE_BITS  "These Bits Enable the appropriate VFD" %
%   N23:86  EV20_OUT_PTR  "EV-20 Rotor Drive Rotor Output Pointer (Selects which VFD is used by EV-3)" %
%   N50:14/10  EV20_ENABLE_CR  "EV-20 Rotor Drive Enable CR" %
%   N61:1  VFD_RUN_BITS_1  "These Bits Initcate the Status Off/Running for the appropriate VFD" %
%   N50:13/10  EV20_RUN  "EV-20 Rotor Drive Running" %
% Rung: 4 %
% This Rung Starts EV-20 Rotor Drive
% when the operator presses the EV-2 PB
% AND
% the Interlocks are satisfied and the motor is Off %
SOR XIC N50:22/6 XIO N50:13/10 XIC N50:3/6 OTL N61:0/[N23:86] EOR
%   N50:22/6  EV20_PB_1S  "EV-20 Rotor Drive On/Off Pushbutton 1-Shot" %
%   N50:13/10  EV20_RUN  "EV-20 Rotor Drive Running" %
%   N50:3/6  EV20_INTERLOCK  "EV-20 Rotor Drive Interlock 0 = Disable 1 = Enable" %
%   N61:0  VFD_ENABLE_BITS  "These Bits Enable the appropriate VFD" %
%   N23:86  EV20_OUT_PTR  "EV-20 Rotor Drive Rotor Output Pointer (Selects which VFD is used by EV-3)" %
% Rung: 5 %
% his Rung Stops EV-20 Rotor Drive
% when the operator presses the EV-2 PB
% AND the motor is ON
% OR
% The Interlocks are NOT satisfied %
SOR BST XIC N50:22/6 XIC N50:13/10 NXB XIO N50:3/6 BND OTU N61:0/[N23:86] EOR
%   N50:22/6  EV20_PB_1S  "EV-20 Rotor Drive On/Off Pushbutton 1-Shot" %
%   N50:13/10  EV20_RUN  "EV-20 Rotor Drive Running" %
%   N50:3/6  EV20_INTERLOCK  "EV-20 Rotor Drive Interlock 0 = Disable 1 = Enable" %
%   N61:0  VFD_ENABLE_BITS  "These Bits Enable the appropriate VFD" %
%   N23:86  EV20_OUT_PTR  "EV-20 Rotor Drive Rotor Output Pointer (Selects which VFD is used by EV-3)" %

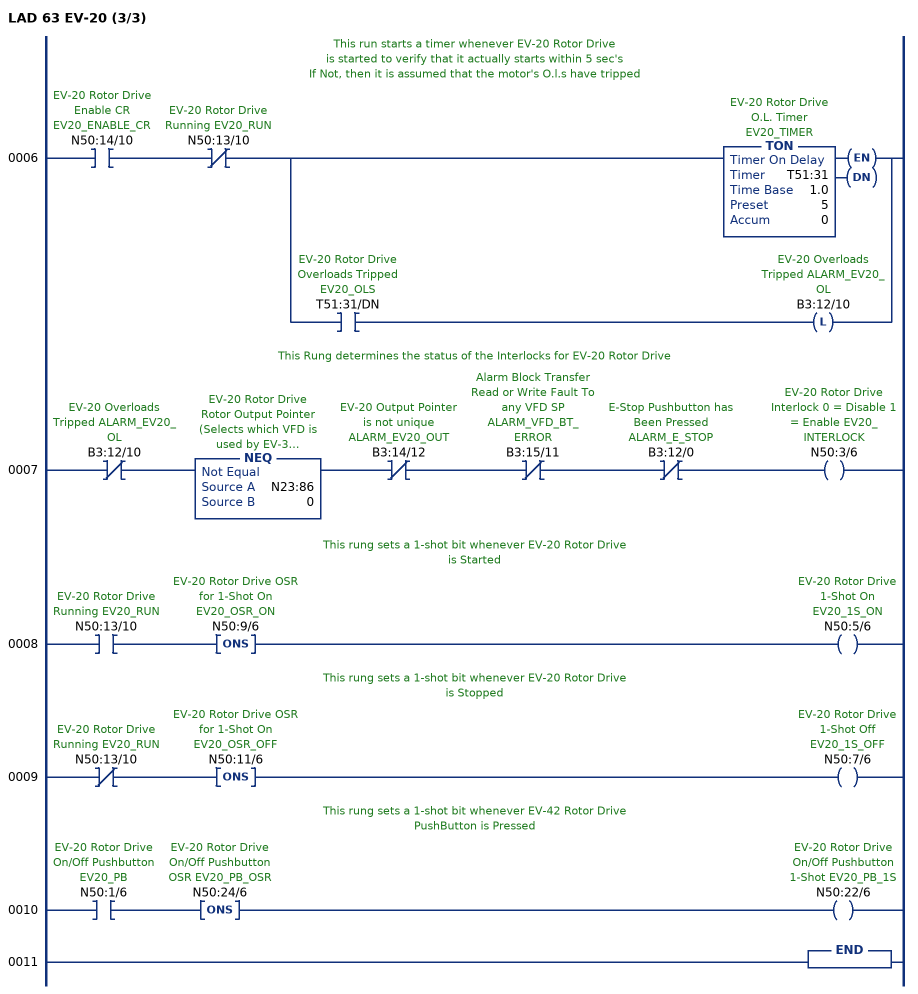
% Rung: 6 %
% This run starts a timer whenever EV-20 Rotor Drive
% is started to verify that it actually starts within 5 sec's
% If Not, then it is assumed that the motor's O.l.s have tripped %
SOR XIC N50:14/10 XIO N50:13/10 BST TON T51:31 1.0 5 0 NXB XIC T51:31/DN OTL B3:12/10 BND EOR
%   N50:14/10  EV20_ENABLE_CR  "EV-20 Rotor Drive Enable CR" %
%   N50:13/10  EV20_RUN  "EV-20 Rotor Drive Running" %
%   T51:31  EV20_TIMER  "EV-20 Rotor Drive O.L. Timer" %
%   T51:31/DN  EV20_OLS  "EV-20 Rotor Drive Overloads Tripped" %
%   B3:12/10  ALARM_EV20_OL  "EV-20 Overloads Tripped" %
% Rung: 7 %
% This Rung determines the status of the Interlocks for EV-20 Rotor Drive %
SOR XIO B3:12/10 NEQ N23:86 0 XIO B3:14/12 XIO B3:15/11 XIO B3:12/0 OTE N50:3/6 EOR
%   B3:12/10  ALARM_EV20_OL  "EV-20 Overloads Tripped" %
%   N23:86  EV20_OUT_PTR  "EV-20 Rotor Drive Rotor Output Pointer (Selects which VFD is used by EV-3)" %
%   B3:14/12  ALARM_EV20_OUT  "EV-20 Output Pointer is not unique" %
%   B3:15/11  ALARM_VFD_BT_ERROR  "Alarm Block Transfer Read or Write Fault To any VFD SP" %
%   B3:12/0  ALARM_E_STOP  "E-Stop Pushbutton has Been Pressed" %
%   N50:3/6  EV20_INTERLOCK  "EV-20 Rotor Drive Interlock 0 = Disable 1 = Enable" %
% Rung: 8 %
% This rung sets a 1-shot bit whenever EV-20 Rotor Drive
% is Started %
SOR XIC N50:13/10 OSR N50:9/6 OTE N50:5/6 EOR
%   N50:13/10  EV20_RUN  "EV-20 Rotor Drive Running" %
%   N50:9/6  EV20_OSR_ON  "EV-20 Rotor Drive OSR for 1-Shot On" %
%   N50:5/6  EV20_1S_ON  "EV-20 Rotor Drive 1-Shot On" %
% Rung: 9 %
% This rung sets a 1-shot bit whenever EV-20 Rotor Drive
% is Stopped %
SOR XIO N50:13/10 OSR N50:11/6 OTE N50:7/6 EOR
%   N50:13/10  EV20_RUN  "EV-20 Rotor Drive Running" %
%   N50:11/6  EV20_OSR_OFF  "EV-20 Rotor Drive OSR for 1-Shot On" %
%   N50:7/6  EV20_1S_OFF  "EV-20 Rotor Drive 1-Shot Off" %
% Rung: 10 %
% This rung sets a 1-shot bit whenever EV-42 Rotor Drive
% PushButton is Pressed %
SOR XIC N50:1/6 OSR N50:24/6 OTE N50:22/6 EOR
%   N50:1/6  EV20_PB  "EV-20 Rotor Drive On/Off Pushbutton" %
%   N50:24/6  EV20_PB_OSR  "EV-20 Rotor Drive On/Off Pushbutton OSR" %
%   N50:22/6  EV20_PB_1S  "EV-20 Rotor Drive On/Off Pushbutton 1-Shot" %
% Rung: 11 %
SOR END EOR

LADDER 64 "PU-21-1"    % PU-21-1 Feed Pump No-1 Controls %
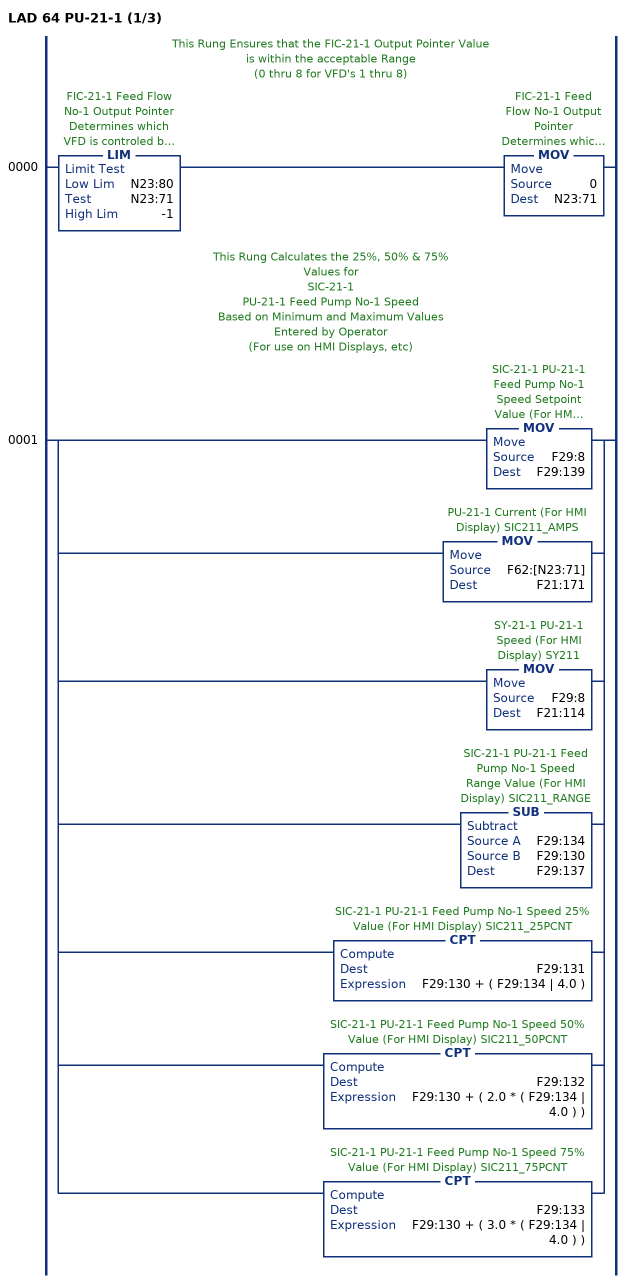
% Rung: 0 %
% This Rung Ensures that the FIC-21-1 Output Pointer Value
% is within the acceptable Range
% (0 thru 8 for VFD's 1 thru 8) %
SOR LIM N23:80 N23:71 -1 MOV 0 N23:71 EOR
%   N23:80  MAX_VFD_ALLOWED_1  "Maximum Number of VFDs Available Plus 1" %
%   N23:71  FIC211_OUT_PTR  "FIC-21-1 Feed Flow No-1 Output Pointer Determines which VFD is controled by FIC" %
% Rung: 1 %
% This Rung Calculates the 25%, 50% & 75%
% Values for
% SIC-21-1
% PU-21-1 Feed Pump No-1 Speed
% Based on Minimum and Maximum Values
% Entered by Operator
% (For use on HMI Displays, etc) %
SOR BST MOV F29:8 F29:139 NXB MOV F62:[N23:71] F21:171 NXB MOV F29:8 F21:114 NXB SUB F29:134 F29:130 F29:137 NXB CPT F29:131 " F29:130 + ( F29:134 | 4.0 ) " NXB CPT F29:132 " F29:130 + ( 2.0 * ( F29:134 | 4.0 ) ) " NXB CPT F29:133 " F29:130 + ( 3.0 * ( F29:134 | 4.0 ) ) " BND EOR
%   F29:8  FIC211_OUT_FP  "FIC-21-1 Output Value (For HMI Display)" %
%   F29:139  SIC211_SP_FP  "SIC-21-1 PU-21-1 Feed Pump No-1 Speed Setpoint Value (For HMI Display)" %
%   N23:71  FIC211_OUT_PTR  "FIC-21-1 Feed Flow No-1 Output Pointer Determines which VFD is controled by FIC" %
%   F21:171  SIC211_AMPS  "PU-21-1 Current (For HMI Display)" %
%   F21:114  SY211  "SY-21-1 PU-21-1 Speed (For HMI Display)" %
%   F29:134  SIC211_MAX  "SIC-21-1 PU-21-1 Feed Pump No-1 Freq at 100% Value (For HMI Display)" %
%   F29:130  SIC211_MIN  "SIC-21-1 PU-21-1 Feed Pump No-1 Speed 0% Value (For HMI Display)" %
%   F29:137  SIC211_RANGE  "SIC-21-1 PU-21-1 Feed Pump No-1 Speed Range Value (For HMI Display)" %
%   F29:131  SIC211_25PCNT  "SIC-21-1 PU-21-1 Feed Pump No-1 Speed 25% Value (For HMI Display)" %
%   F29:132  SIC211_50PCNT  "SIC-21-1 PU-21-1 Feed Pump No-1 Speed 50% Value (For HMI Display)" %
%   F29:133  SIC211_75PCNT  "SIC-21-1 PU-21-1 Feed Pump No-1 Speed 75% Value (For HMI Display)" %

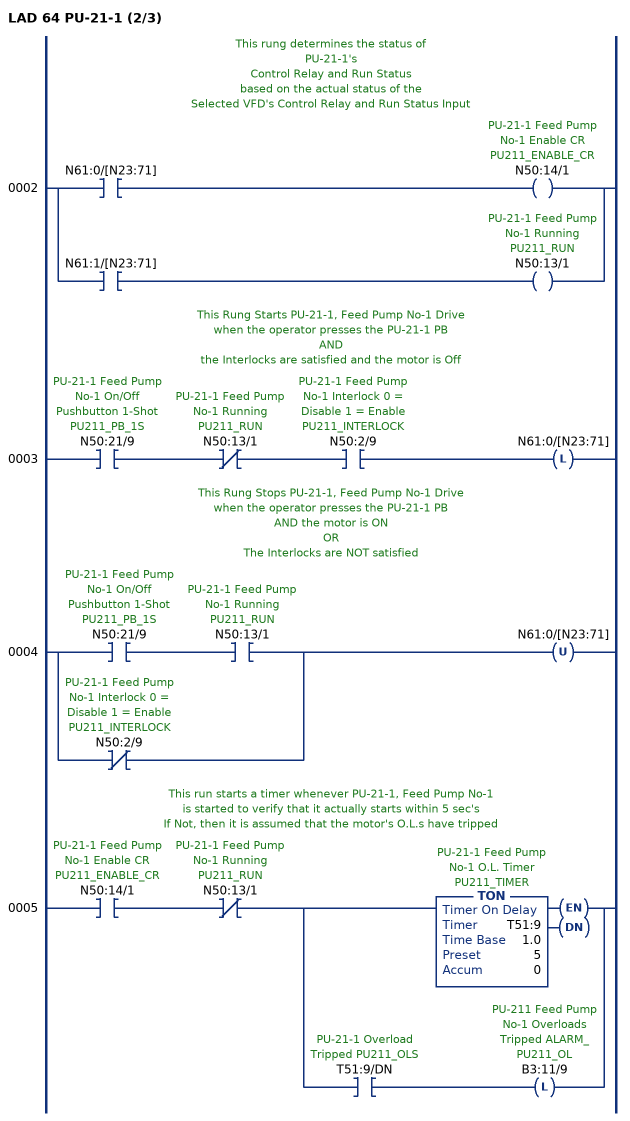
% Rung: 2 %
% This rung determines the status of
% PU-21-1's
% Control Relay and Run Status
% based on the actual status of the
% Selected VFD's Control Relay and Run Status Input %
SOR BST XIC N61:0/[N23:71] OTE N50:14/1 NXB XIC N61:1/[N23:71] OTE N50:13/1 BND EOR
%   N61:0  VFD_ENABLE_BITS  "These Bits Enable the appropriate VFD" %
%   N23:71  FIC211_OUT_PTR  "FIC-21-1 Feed Flow No-1 Output Pointer Determines which VFD is controled by FIC" %
%   N50:14/1  PU211_ENABLE_CR  "PU-21-1 Feed Pump No-1 Enable CR" %
%   N61:1  VFD_RUN_BITS_1  "These Bits Initcate the Status Off/Running for the appropriate VFD" %
%   N50:13/1  PU211_RUN  "PU-21-1 Feed Pump No-1 Running" %
% Rung: 3 %
% This Rung Starts PU-21-1, Feed Pump No-1 Drive
% when the operator presses the PU-21-1 PB
% AND
% the Interlocks are satisfied and the motor is Off %
SOR XIC N50:21/9 XIO N50:13/1 XIC N50:2/9 OTL N61:0/[N23:71] EOR
%   N50:21/9  PU211_PB_1S  "PU-21-1 Feed Pump No-1 On/Off Pushbutton 1-Shot" %
%   N50:13/1  PU211_RUN  "PU-21-1 Feed Pump No-1 Running" %
%   N50:2/9  PU211_INTERLOCK  "PU-21-1 Feed Pump No-1 Interlock 0 = Disable 1 = Enable" %
%   N61:0  VFD_ENABLE_BITS  "These Bits Enable the appropriate VFD" %
%   N23:71  FIC211_OUT_PTR  "FIC-21-1 Feed Flow No-1 Output Pointer Determines which VFD is controled by FIC" %
% Rung: 4 %
% This Rung Stops PU-21-1, Feed Pump No-1 Drive
% when the operator presses the PU-21-1 PB
% AND the motor is ON
% OR
% The Interlocks are NOT satisfied %
SOR BST XIC N50:21/9 XIC N50:13/1 NXB XIO N50:2/9 BND OTU N61:0/[N23:71] EOR
%   N50:21/9  PU211_PB_1S  "PU-21-1 Feed Pump No-1 On/Off Pushbutton 1-Shot" %
%   N50:13/1  PU211_RUN  "PU-21-1 Feed Pump No-1 Running" %
%   N50:2/9  PU211_INTERLOCK  "PU-21-1 Feed Pump No-1 Interlock 0 = Disable 1 = Enable" %
%   N61:0  VFD_ENABLE_BITS  "These Bits Enable the appropriate VFD" %
%   N23:71  FIC211_OUT_PTR  "FIC-21-1 Feed Flow No-1 Output Pointer Determines which VFD is controled by FIC" %
% Rung: 5 %
% This run starts a timer whenever PU-21-1, Feed Pump No-1
% is started to verify that it actually starts within 5 sec's
% If Not, then it is assumed that the motor's O.L.s have tripped %
SOR XIC N50:14/1 XIO N50:13/1 BST TON T51:9 1.0 5 0 NXB XIC T51:9/DN OTL B3:11/9 BND EOR
%   N50:14/1  PU211_ENABLE_CR  "PU-21-1 Feed Pump No-1 Enable CR" %
%   N50:13/1  PU211_RUN  "PU-21-1 Feed Pump No-1 Running" %
%   T51:9  PU211_TIMER  "PU-21-1 Feed Pump No-1 O.L. Timer" %
%   T51:9/DN  PU211_OLS  "PU-21-1 Overload Tripped" %
%   B3:11/9  ALARM_PU211_OL  "PU-211 Feed Pump No-1 Overloads Tripped" %

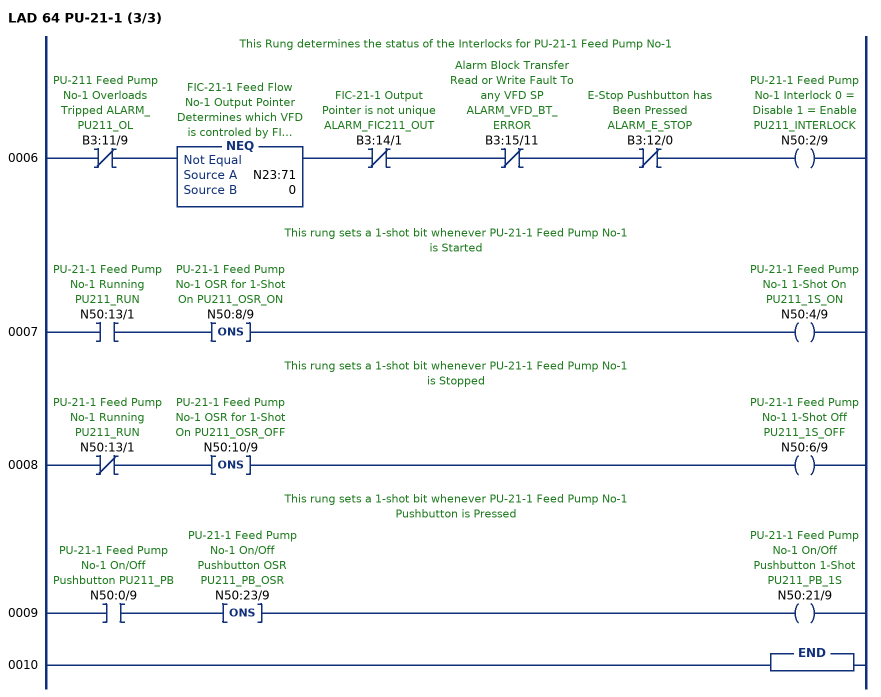
% Rung: 6 %
% This Rung determines the status of the Interlocks for PU-21-1 Feed Pump No-1 %
SOR XIO B3:11/9 NEQ N23:71 0 XIO B3:14/1 XIO B3:15/11 XIO B3:12/0 OTE N50:2/9 EOR
%   B3:11/9  ALARM_PU211_OL  "PU-211 Feed Pump No-1 Overloads Tripped" %
%   N23:71  FIC211_OUT_PTR  "FIC-21-1 Feed Flow No-1 Output Pointer Determines which VFD is controled by FIC" %
%   B3:14/1  ALARM_FIC211_OUT  "FIC-21-1 Output Pointer is not unique" %
%   B3:15/11  ALARM_VFD_BT_ERROR  "Alarm Block Transfer Read or Write Fault To any VFD SP" %
%   B3:12/0  ALARM_E_STOP  "E-Stop Pushbutton has Been Pressed" %
%   N50:2/9  PU211_INTERLOCK  "PU-21-1 Feed Pump No-1 Interlock 0 = Disable 1 = Enable" %
% Rung: 7 %
% This rung sets a 1-shot bit whenever PU-21-1 Feed Pump No-1
% is Started %
SOR XIC N50:13/1 OSR N50:8/9 OTE N50:4/9 EOR
%   N50:13/1  PU211_RUN  "PU-21-1 Feed Pump No-1 Running" %
%   N50:8/9  PU211_OSR_ON  "PU-21-1 Feed Pump No-1 OSR for 1-Shot On" %
%   N50:4/9  PU211_1S_ON  "PU-21-1 Feed Pump No-1 1-Shot On" %
% Rung: 8 %
% This rung sets a 1-shot bit whenever PU-21-1 Feed Pump No-1
% is Stopped %
SOR XIO N50:13/1 OSR N50:10/9 OTE N50:6/9 EOR
%   N50:13/1  PU211_RUN  "PU-21-1 Feed Pump No-1 Running" %
%   N50:10/9  PU211_OSR_OFF  "PU-21-1 Feed Pump No-1 OSR for 1-Shot On" %
%   N50:6/9  PU211_1S_OFF  "PU-21-1 Feed Pump No-1 1-Shot Off" %
% Rung: 9 %
% This rung sets a 1-shot bit whenever PU-21-1 Feed Pump No-1
% Pushbutton is Pressed %
SOR XIC N50:0/9 OSR N50:23/9 OTE N50:21/9 EOR
%   N50:0/9  PU211_PB  "PU-21-1 Feed Pump No-1 On/Off Pushbutton" %
%   N50:23/9  PU211_PB_OSR  "PU-21-1 Feed Pump No-1 On/Off Pushbutton OSR" %
%   N50:21/9  PU211_PB_1S  "PU-21-1 Feed Pump No-1 On/Off Pushbutton 1-Shot" %
% Rung: 10 %
SOR END EOR

LADDER 65 "PU-21-2"    % PU-21-2 Feed Pump No-2 Controls %
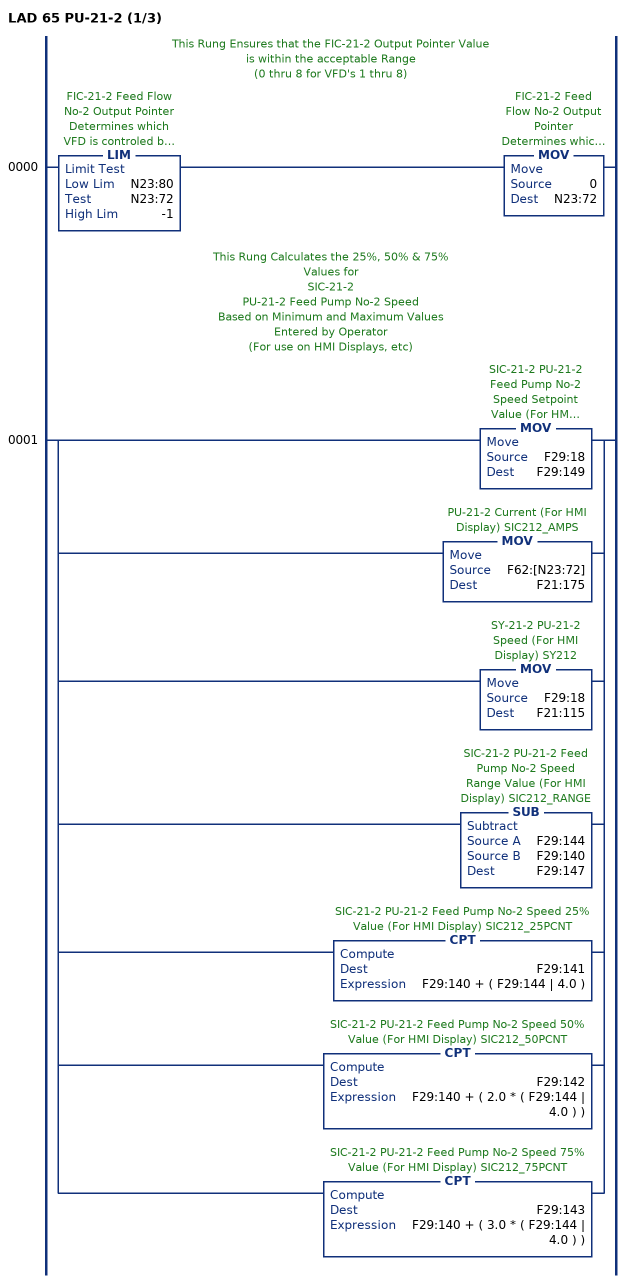
% Rung: 0 %
% This Rung Ensures that the FIC-21-2 Output Pointer Value
% is within the acceptable Range
% (0 thru 8 for VFD's 1 thru 8) %
SOR LIM N23:80 N23:72 -1 MOV 0 N23:72 EOR
%   N23:80  MAX_VFD_ALLOWED_1  "Maximum Number of VFDs Available Plus 1" %
%   N23:72  FIC212_OUT_PTR  "FIC-21-2 Feed Flow No-2 Output Pointer Determines which VFD is controled by FIC" %
% Rung: 1 %
% This Rung Calculates the 25%, 50% & 75%
% Values for
% SIC-21-2
% PU-21-2 Feed Pump No-2 Speed
% Based on Minimum and Maximum Values
% Entered by Operator
% (For use on HMI Displays, etc) %
SOR BST MOV F29:18 F29:149 NXB MOV F62:[N23:72] F21:175 NXB MOV F29:18 F21:115 NXB SUB F29:144 F29:140 F29:147 NXB CPT F29:141 " F29:140 + ( F29:144 | 4.0 ) " NXB CPT F29:142 " F29:140 + ( 2.0 * ( F29:144 | 4.0 ) ) " NXB CPT F29:143 " F29:140 + ( 3.0 * ( F29:144 | 4.0 ) ) " BND EOR
%   F29:18  FIC212_OUT_FP  "FIC-21-2 Output Value (For HMI Display)" %
%   F29:149  SIC212_SP_FP  "SIC-21-2 PU-21-2 Feed Pump No-2 Speed Setpoint Value (For HMI Display)" %
%   N23:72  FIC212_OUT_PTR  "FIC-21-2 Feed Flow No-2 Output Pointer Determines which VFD is controled by FIC" %
%   F21:175  SIC212_AMPS  "PU-21-2 Current (For HMI Display)" %
%   F21:115  SY212  "SY-21-2 PU-21-2 Speed (For HMI Display)" %
%   F29:144  SIC212_MAX  "SIC-21-2 PU-21-2 Feed Pump No-2 Freq at 100% Value (For HMI Display)" %
%   F29:140  SIC212_MIN  "SIC-21-2 PU-21-2 Feed Pump No-2 Speed 0% Value (For HMI Display)" %
%   F29:147  SIC212_RANGE  "SIC-21-2 PU-21-2 Feed Pump No-2 Speed Range Value (For HMI Display)" %
%   F29:141  SIC212_25PCNT  "SIC-21-2 PU-21-2 Feed Pump No-2 Speed 25% Value (For HMI Display)" %
%   F29:142  SIC212_50PCNT  "SIC-21-2 PU-21-2 Feed Pump No-2 Speed 50% Value (For HMI Display)" %
%   F29:143  SIC212_75PCNT  "SIC-21-2 PU-21-2 Feed Pump No-2 Speed 75% Value (For HMI Display)" %

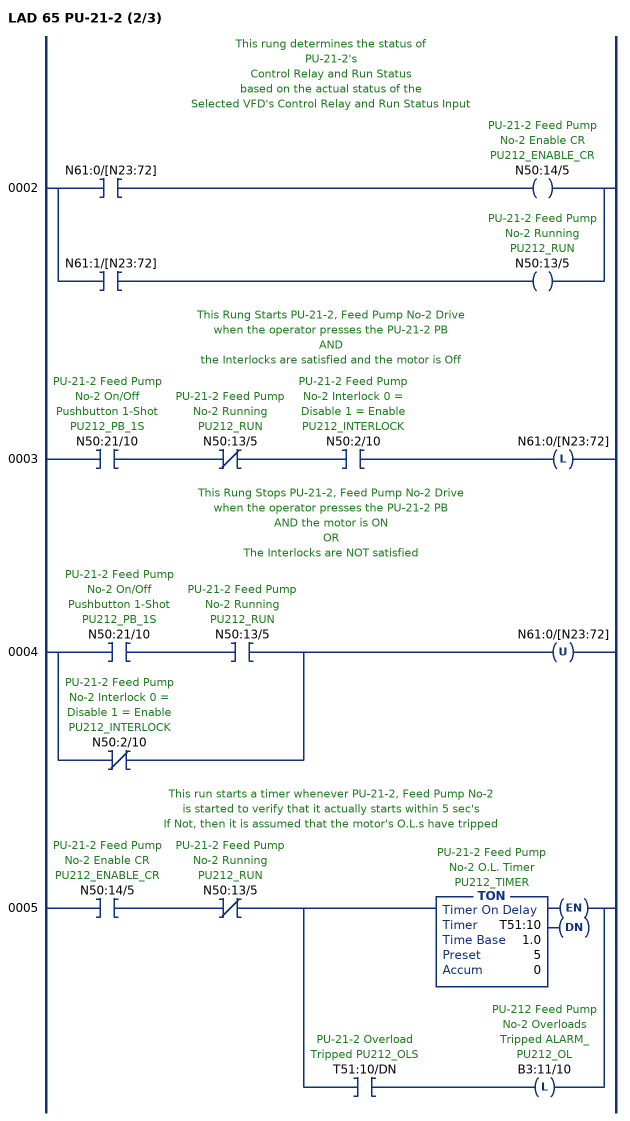
% Rung: 2 %
% This rung determines the status of
% PU-21-2's
% Control Relay and Run Status
% based on the actual status of the
% Selected VFD's Control Relay and Run Status Input %
SOR BST XIC N61:0/[N23:72] OTE N50:14/5 NXB XIC N61:1/[N23:72] OTE N50:13/5 BND EOR
%   N61:0  VFD_ENABLE_BITS  "These Bits Enable the appropriate VFD" %
%   N23:72  FIC212_OUT_PTR  "FIC-21-2 Feed Flow No-2 Output Pointer Determines which VFD is controled by FIC" %
%   N50:14/5  PU212_ENABLE_CR  "PU-21-2 Feed Pump No-2 Enable CR" %
%   N61:1  VFD_RUN_BITS_1  "These Bits Initcate the Status Off/Running for the appropriate VFD" %
%   N50:13/5  PU212_RUN  "PU-21-2 Feed Pump No-2 Running" %
% Rung: 3 %
% This Rung Starts PU-21-2, Feed Pump No-2 Drive
% when the operator presses the PU-21-2 PB
% AND
% the Interlocks are satisfied and the motor is Off %
SOR XIC N50:21/10 XIO N50:13/5 XIC N50:2/10 OTL N61:0/[N23:72] EOR
%   N50:21/10  PU212_PB_1S  "PU-21-2 Feed Pump No-2 On/Off Pushbutton 1-Shot" %
%   N50:13/5  PU212_RUN  "PU-21-2 Feed Pump No-2 Running" %
%   N50:2/10  PU212_INTERLOCK  "PU-21-2 Feed Pump No-2 Interlock 0 = Disable 1 = Enable" %
%   N61:0  VFD_ENABLE_BITS  "These Bits Enable the appropriate VFD" %
%   N23:72  FIC212_OUT_PTR  "FIC-21-2 Feed Flow No-2 Output Pointer Determines which VFD is controled by FIC" %
% Rung: 4 %
% This Rung Stops PU-21-2, Feed Pump No-2 Drive
% when the operator presses the PU-21-2 PB
% AND the motor is ON
% OR
% The Interlocks are NOT satisfied %
SOR BST XIC N50:21/10 XIC N50:13/5 NXB XIO N50:2/10 BND OTU N61:0/[N23:72] EOR
%   N50:21/10  PU212_PB_1S  "PU-21-2 Feed Pump No-2 On/Off Pushbutton 1-Shot" %
%   N50:13/5  PU212_RUN  "PU-21-2 Feed Pump No-2 Running" %
%   N50:2/10  PU212_INTERLOCK  "PU-21-2 Feed Pump No-2 Interlock 0 = Disable 1 = Enable" %
%   N61:0  VFD_ENABLE_BITS  "These Bits Enable the appropriate VFD" %
%   N23:72  FIC212_OUT_PTR  "FIC-21-2 Feed Flow No-2 Output Pointer Determines which VFD is controled by FIC" %
% Rung: 5 %
% This run starts a timer whenever PU-21-2, Feed Pump No-2
% is started to verify that it actually starts within 5 sec's
% If Not, then it is assumed that the motor's O.L.s have tripped %
SOR XIC N50:14/5 XIO N50:13/5 BST TON T51:10 1.0 5 0 NXB XIC T51:10/DN OTL B3:11/10 BND EOR
%   N50:14/5  PU212_ENABLE_CR  "PU-21-2 Feed Pump No-2 Enable CR" %
%   N50:13/5  PU212_RUN  "PU-21-2 Feed Pump No-2 Running" %
%   T51:10  PU212_TIMER  "PU-21-2 Feed Pump No-2 O.L. Timer" %
%   T51:10/DN  PU212_OLS  "PU-21-2 Overload Tripped" %
%   B3:11/10  ALARM_PU212_OL  "PU-212 Feed Pump No-2 Overloads Tripped" %

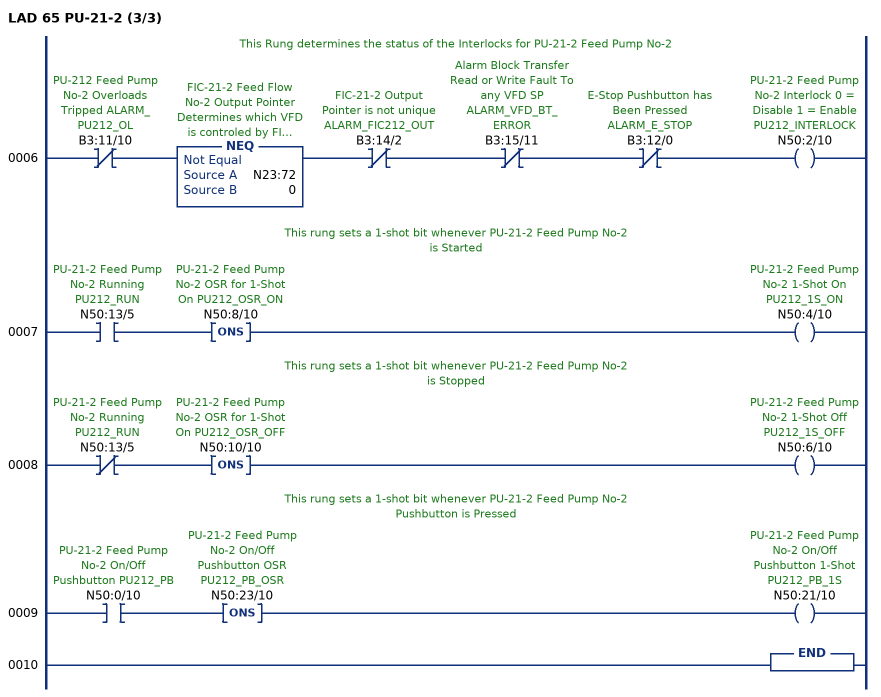
% Rung: 6 %
% This Rung determines the status of the Interlocks for PU-21-2 Feed Pump No-2 %
SOR XIO B3:11/10 NEQ N23:72 0 XIO B3:14/2 XIO B3:15/11 XIO B3:12/0 OTE N50:2/10 EOR
%   B3:11/10  ALARM_PU212_OL  "PU-212 Feed Pump No-2 Overloads Tripped" %
%   N23:72  FIC212_OUT_PTR  "FIC-21-2 Feed Flow No-2 Output Pointer Determines which VFD is controled by FIC" %
%   B3:14/2  ALARM_FIC212_OUT  "FIC-21-2 Output Pointer is not unique" %
%   B3:15/11  ALARM_VFD_BT_ERROR  "Alarm Block Transfer Read or Write Fault To any VFD SP" %
%   B3:12/0  ALARM_E_STOP  "E-Stop Pushbutton has Been Pressed" %
%   N50:2/10  PU212_INTERLOCK  "PU-21-2 Feed Pump No-2 Interlock 0 = Disable 1 = Enable" %
% Rung: 7 %
% This rung sets a 1-shot bit whenever PU-21-2 Feed Pump No-2
% is Started %
SOR XIC N50:13/5 OSR N50:8/10 OTE N50:4/10 EOR
%   N50:13/5  PU212_RUN  "PU-21-2 Feed Pump No-2 Running" %
%   N50:8/10  PU212_OSR_ON  "PU-21-2 Feed Pump No-2 OSR for 1-Shot On" %
%   N50:4/10  PU212_1S_ON  "PU-21-2 Feed Pump No-2 1-Shot On" %
% Rung: 8 %
% This rung sets a 1-shot bit whenever PU-21-2 Feed Pump No-2
% is Stopped %
SOR XIO N50:13/5 OSR N50:10/10 OTE N50:6/10 EOR
%   N50:13/5  PU212_RUN  "PU-21-2 Feed Pump No-2 Running" %
%   N50:10/10  PU212_OSR_OFF  "PU-21-2 Feed Pump No-2 OSR for 1-Shot On" %
%   N50:6/10  PU212_1S_OFF  "PU-21-2 Feed Pump No-2 1-Shot Off" %
% Rung: 9 %
% This rung sets a 1-shot bit whenever PU-21-2 Feed Pump No-2
% Pushbutton is Pressed %
SOR XIC N50:0/10 OSR N50:23/10 OTE N50:21/10 EOR
%   N50:0/10  PU212_PB  "PU-21-2 Feed Pump No-2 On/Off Pushbutton" %
%   N50:23/10  PU212_PB_OSR  "PU-21-2 Feed Pump No-2 On/Off Pushbutton OSR" %
%   N50:21/10  PU212_PB_1S  "PU-21-2 Feed Pump No-2 On/Off Pushbutton 1-Shot" %
% Rung: 10 %
SOR END EOR

LADDER 66 "PU-21-3"    % PU-21-3 Feed Pump No-3 Controls %
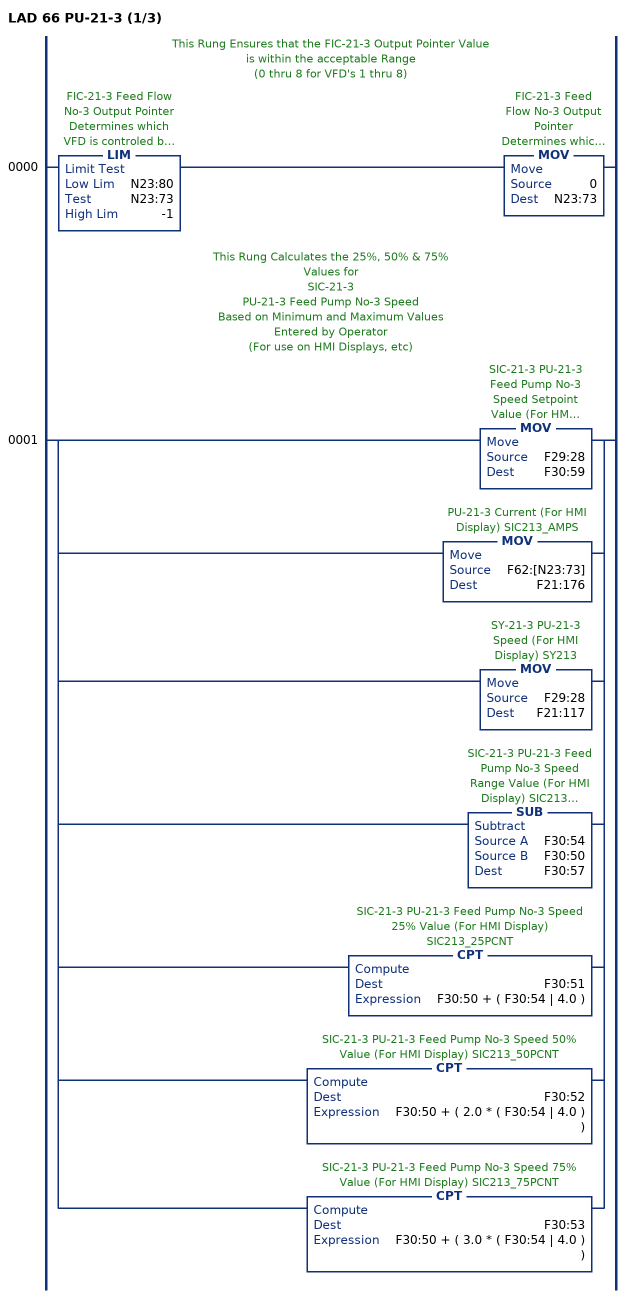
% Rung: 0 %
% This Rung Ensures that the FIC-21-3 Output Pointer Value
% is within the acceptable Range
% (0 thru 8 for VFD's 1 thru 8) %
SOR LIM N23:80 N23:73 -1 MOV 0 N23:73 EOR
%   N23:80  MAX_VFD_ALLOWED_1  "Maximum Number of VFDs Available Plus 1" %
%   N23:73  FIC213_OUT_PTR  "FIC-21-3 Feed Flow No-3 Output Pointer Determines which VFD is controled by FIC" %
% Rung: 1 %
% This Rung Calculates the 25%, 50% & 75%
% Values for
% SIC-21-3
% PU-21-3 Feed Pump No-3 Speed
% Based on Minimum and Maximum Values
% Entered by Operator
% (For use on HMI Displays, etc) %
SOR BST MOV F29:28 F30:59 NXB MOV F62:[N23:73] F21:176 NXB MOV F29:28 F21:117 NXB SUB F30:54 F30:50 F30:57 NXB CPT F30:51 " F30:50 + ( F30:54 | 4.0 ) " NXB CPT F30:52 " F30:50 + ( 2.0 * ( F30:54 | 4.0 ) ) " NXB CPT F30:53 " F30:50 + ( 3.0 * ( F30:54 | 4.0 ) ) " BND EOR
%   F29:28  FIC213_OUT_FP  "FIC-21-3 Output Value (For HMI Display)" %
%   F30:59  SIC213_SP_FP  "SIC-21-3 PU-21-3 Feed Pump No-3 Speed Setpoint Value (For HMI Display)" %
%   N23:73  FIC213_OUT_PTR  "FIC-21-3 Feed Flow No-3 Output Pointer Determines which VFD is controled by FIC" %
%   F21:176  SIC213_AMPS  "PU-21-3 Current (For HMI Display)" %
%   F21:117  SY213  "SY-21-3 PU-21-3 Speed (For HMI Display)" %
%   F30:54  SIC213_MAX  "SIC-21-3 PU-21-3 Feed Pump No-3 Freq at 100% Value (For HMI Display)" %
%   F30:50  SIC213_MIN  "SIC-21-3 PU-21-3 Feed Pump No-3 Speed 0% Value (For HMI Display)" %
%   F30:57  SIC213_RANGE  "SIC-21-3 PU-21-3 Feed Pump No-3 Speed Range Value (For HMI Display)" %
%   F30:51  SIC213_25PCNT  "SIC-21-3 PU-21-3 Feed Pump No-3 Speed 25% Value (For HMI Display)" %
%   F30:52  SIC213_50PCNT  "SIC-21-3 PU-21-3 Feed Pump No-3 Speed 50% Value (For HMI Display)" %
%   F30:53  SIC213_75PCNT  "SIC-21-3 PU-21-3 Feed Pump No-3 Speed 75% Value (For HMI Display)" %

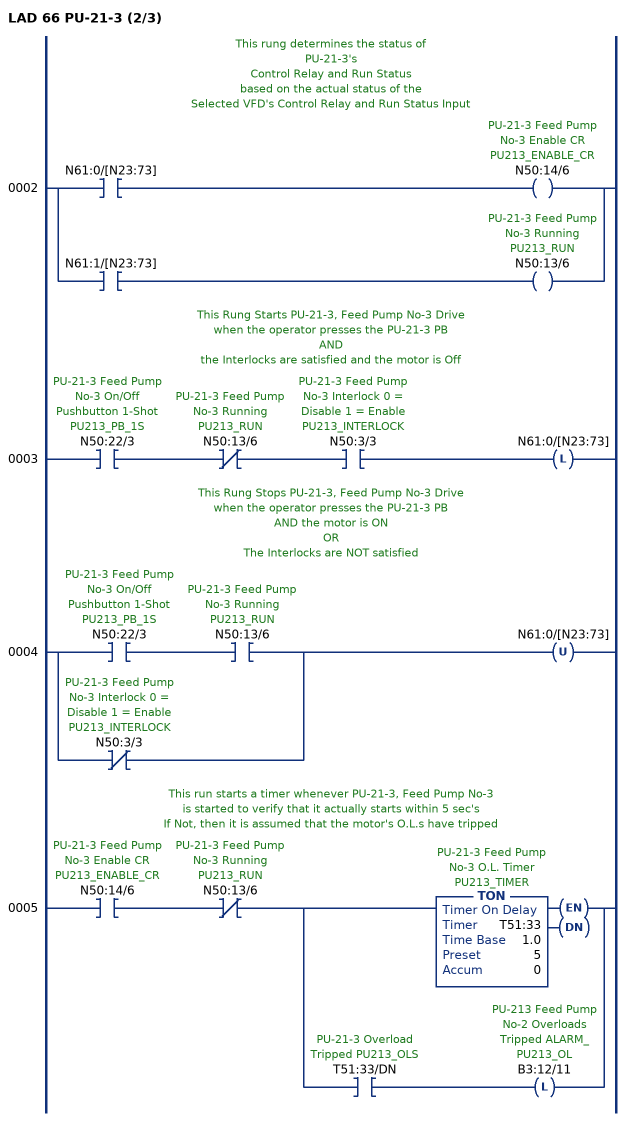
% Rung: 2 %
% This rung determines the status of
% PU-21-3's
% Control Relay and Run Status
% based on the actual status of the
% Selected VFD's Control Relay and Run Status Input %
SOR BST XIC N61:0/[N23:73] OTE N50:14/6 NXB XIC N61:1/[N23:73] OTE N50:13/6 BND EOR
%   N61:0  VFD_ENABLE_BITS  "These Bits Enable the appropriate VFD" %
%   N23:73  FIC213_OUT_PTR  "FIC-21-3 Feed Flow No-3 Output Pointer Determines which VFD is controled by FIC" %
%   N50:14/6  PU213_ENABLE_CR  "PU-21-3 Feed Pump No-3 Enable CR" %
%   N61:1  VFD_RUN_BITS_1  "These Bits Initcate the Status Off/Running for the appropriate VFD" %
%   N50:13/6  PU213_RUN  "PU-21-3 Feed Pump No-3 Running" %
% Rung: 3 %
% This Rung Starts PU-21-3, Feed Pump No-3 Drive
% when the operator presses the PU-21-3 PB
% AND
% the Interlocks are satisfied and the motor is Off %
SOR XIC N50:22/3 XIO N50:13/6 XIC N50:3/3 OTL N61:0/[N23:73] EOR
%   N50:22/3  PU213_PB_1S  "PU-21-3 Feed Pump No-3 On/Off Pushbutton 1-Shot" %
%   N50:13/6  PU213_RUN  "PU-21-3 Feed Pump No-3 Running" %
%   N50:3/3  PU213_INTERLOCK  "PU-21-3 Feed Pump No-3 Interlock 0 = Disable 1 = Enable" %
%   N61:0  VFD_ENABLE_BITS  "These Bits Enable the appropriate VFD" %
%   N23:73  FIC213_OUT_PTR  "FIC-21-3 Feed Flow No-3 Output Pointer Determines which VFD is controled by FIC" %
% Rung: 4 %
% This Rung Stops PU-21-3, Feed Pump No-3 Drive
% when the operator presses the PU-21-3 PB
% AND the motor is ON
% OR
% The Interlocks are NOT satisfied %
SOR BST XIC N50:22/3 XIC N50:13/6 NXB XIO N50:3/3 BND OTU N61:0/[N23:73] EOR
%   N50:22/3  PU213_PB_1S  "PU-21-3 Feed Pump No-3 On/Off Pushbutton 1-Shot" %
%   N50:13/6  PU213_RUN  "PU-21-3 Feed Pump No-3 Running" %
%   N50:3/3  PU213_INTERLOCK  "PU-21-3 Feed Pump No-3 Interlock 0 = Disable 1 = Enable" %
%   N61:0  VFD_ENABLE_BITS  "These Bits Enable the appropriate VFD" %
%   N23:73  FIC213_OUT_PTR  "FIC-21-3 Feed Flow No-3 Output Pointer Determines which VFD is controled by FIC" %
% Rung: 5 %
% This run starts a timer whenever PU-21-3, Feed Pump No-3
% is started to verify that it actually starts within 5 sec's
% If Not, then it is assumed that the motor's O.L.s have tripped %
SOR XIC N50:14/6 XIO N50:13/6 BST TON T51:33 1.0 5 0 NXB XIC T51:33/DN OTL B3:12/11 BND EOR
%   N50:14/6  PU213_ENABLE_CR  "PU-21-3 Feed Pump No-3 Enable CR" %
%   N50:13/6  PU213_RUN  "PU-21-3 Feed Pump No-3 Running" %
%   T51:33  PU213_TIMER  "PU-21-3 Feed Pump No-3 O.L. Timer" %
%   T51:33/DN  PU213_OLS  "PU-21-3 Overload Tripped" %
%   B3:12/11  ALARM_PU213_OL  "PU-213 Feed Pump No-2 Overloads Tripped" %

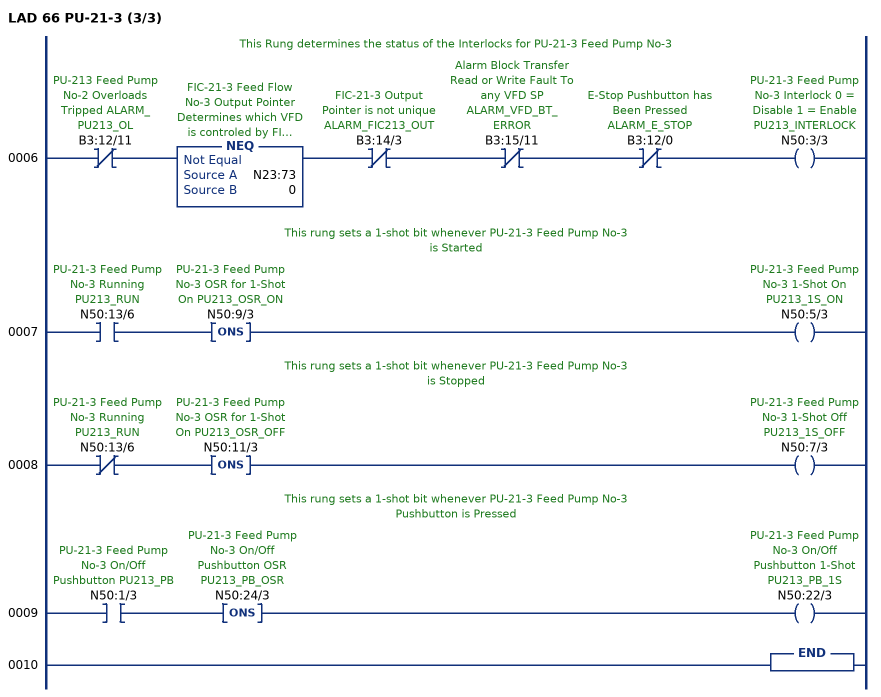
% Rung: 6 %
% This Rung determines the status of the Interlocks for PU-21-3 Feed Pump No-3 %
SOR XIO B3:12/11 NEQ N23:73 0 XIO B3:14/3 XIO B3:15/11 XIO B3:12/0 OTE N50:3/3 EOR
%   B3:12/11  ALARM_PU213_OL  "PU-213 Feed Pump No-2 Overloads Tripped" %
%   N23:73  FIC213_OUT_PTR  "FIC-21-3 Feed Flow No-3 Output Pointer Determines which VFD is controled by FIC" %
%   B3:14/3  ALARM_FIC213_OUT  "FIC-21-3 Output Pointer is not unique" %
%   B3:15/11  ALARM_VFD_BT_ERROR  "Alarm Block Transfer Read or Write Fault To any VFD SP" %
%   B3:12/0  ALARM_E_STOP  "E-Stop Pushbutton has Been Pressed" %
%   N50:3/3  PU213_INTERLOCK  "PU-21-3 Feed Pump No-3 Interlock 0 = Disable 1 = Enable" %
% Rung: 7 %
% This rung sets a 1-shot bit whenever PU-21-3 Feed Pump No-3
% is Started %
SOR XIC N50:13/6 OSR N50:9/3 OTE N50:5/3 EOR
%   N50:13/6  PU213_RUN  "PU-21-3 Feed Pump No-3 Running" %
%   N50:9/3  PU213_OSR_ON  "PU-21-3 Feed Pump No-3 OSR for 1-Shot On" %
%   N50:5/3  PU213_1S_ON  "PU-21-3 Feed Pump No-3 1-Shot On" %
% Rung: 8 %
% This rung sets a 1-shot bit whenever PU-21-3 Feed Pump No-3
% is Stopped %
SOR XIO N50:13/6 OSR N50:11/3 OTE N50:7/3 EOR
%   N50:13/6  PU213_RUN  "PU-21-3 Feed Pump No-3 Running" %
%   N50:11/3  PU213_OSR_OFF  "PU-21-3 Feed Pump No-3 OSR for 1-Shot On" %
%   N50:7/3  PU213_1S_OFF  "PU-21-3 Feed Pump No-3 1-Shot Off" %
% Rung: 9 %
% This rung sets a 1-shot bit whenever PU-21-3 Feed Pump No-3
% Pushbutton is Pressed %
SOR XIC N50:1/3 OSR N50:24/3 OTE N50:22/3 EOR
%   N50:1/3  PU213_PB  "PU-21-3 Feed Pump No-3 On/Off Pushbutton" %
%   N50:24/3  PU213_PB_OSR  "PU-21-3 Feed Pump No-3 On/Off Pushbutton OSR" %
%   N50:22/3  PU213_PB_1S  "PU-21-3 Feed Pump No-3 On/Off Pushbutton 1-Shot" %
% Rung: 10 %
SOR END EOR

LADDER 67 "PU-21-4"    % PU-21-4 Feed Pump No-4 Controls %
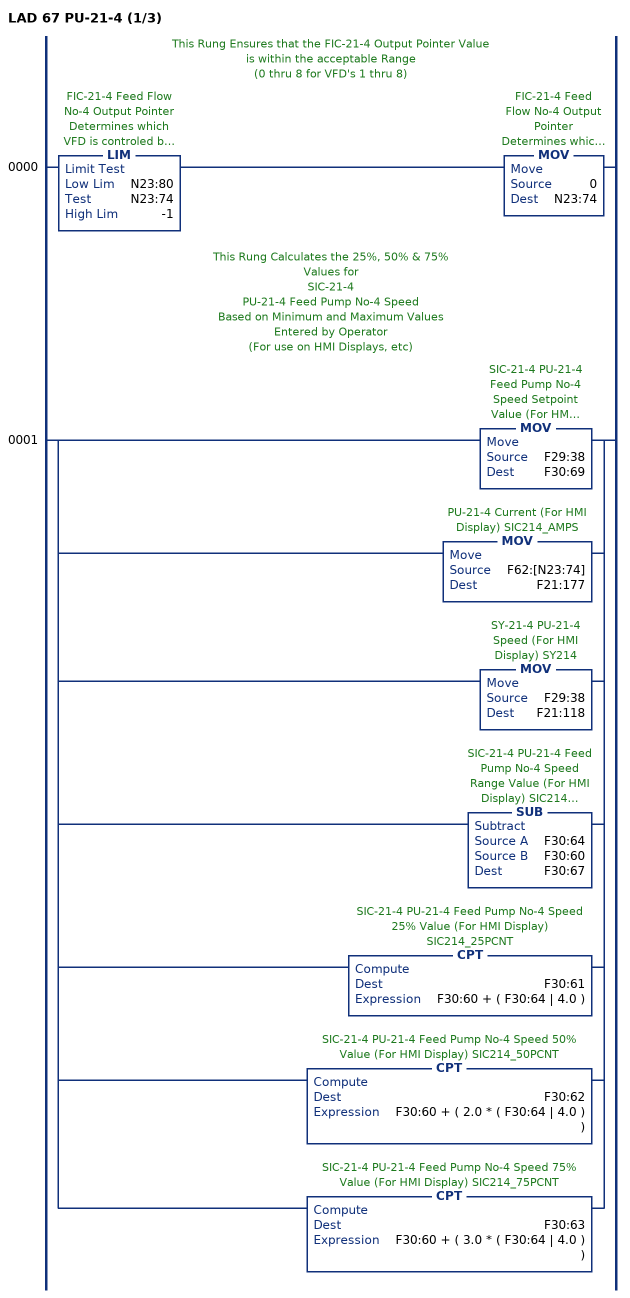
% Rung: 0 %
% This Rung Ensures that the FIC-21-4 Output Pointer Value
% is within the acceptable Range
% (0 thru 8 for VFD's 1 thru 8) %
SOR LIM N23:80 N23:74 -1 MOV 0 N23:74 EOR
%   N23:80  MAX_VFD_ALLOWED_1  "Maximum Number of VFDs Available Plus 1" %
%   N23:74  FIC214_OUT_PTR  "FIC-21-4 Feed Flow No-4 Output Pointer Determines which VFD is controled by FIC" %
% Rung: 1 %
% This Rung Calculates the 25%, 50% & 75%
% Values for
% SIC-21-4
% PU-21-4 Feed Pump No-4 Speed
% Based on Minimum and Maximum Values
% Entered by Operator
% (For use on HMI Displays, etc) %
SOR BST MOV F29:38 F30:69 NXB MOV F62:[N23:74] F21:177 NXB MOV F29:38 F21:118 NXB SUB F30:64 F30:60 F30:67 NXB CPT F30:61 " F30:60 + ( F30:64 | 4.0 ) " NXB CPT F30:62 " F30:60 + ( 2.0 * ( F30:64 | 4.0 ) ) " NXB CPT F30:63 " F30:60 + ( 3.0 * ( F30:64 | 4.0 ) ) " BND EOR
%   F29:38  FIC214_OUT_FP  "FIC-21-4 Output Value (For HMI Display)" %
%   F30:69  SIC214_SP_FP  "SIC-21-4 PU-21-4 Feed Pump No-4 Speed Setpoint Value (For HMI Display)" %
%   N23:74  FIC214_OUT_PTR  "FIC-21-4 Feed Flow No-4 Output Pointer Determines which VFD is controled by FIC" %
%   F21:177  SIC214_AMPS  "PU-21-4 Current (For HMI Display)" %
%   F21:118  SY214  "SY-21-4 PU-21-4 Speed (For HMI Display)" %
%   F30:64  SIC214_MAX  "SIC-21-4 PU-21-4 Feed Pump No-4 Freq at 100% Value (For HMI Display)" %
%   F30:60  SIC214_MIN  "SIC-21-4 PU-21-4 Feed Pump No-4 Speed 0% Value (For HMI Display)" %
%   F30:67  SIC214_RANGE  "SIC-21-4 PU-21-4 Feed Pump No-4 Speed Range Value (For HMI Display)" %
%   F30:61  SIC214_25PCNT  "SIC-21-4 PU-21-4 Feed Pump No-4 Speed 25% Value (For HMI Display)" %
%   F30:62  SIC214_50PCNT  "SIC-21-4 PU-21-4 Feed Pump No-4 Speed 50% Value (For HMI Display)" %
%   F30:63  SIC214_75PCNT  "SIC-21-4 PU-21-4 Feed Pump No-4 Speed 75% Value (For HMI Display)" %

